LIN {X 0,Y 516.566,Z 410.559,A -85,B 0,C 180,E1 -4941.393,E2 -4941.393} C_VEL
LIN {X 0,Y 516.57,Z 414.408,A -85,B 0,C 180,E1 -4943.752,E2 -4943.752} C_VEL
LIN {X 0,Y 516.545,Z 418.324,A -85,B 0,C 180,E1 -4946.099,E2 -4946.099} C_VEL
LIN {X 0,Y 516.317,Z 423.538,A -85,B 0,C 180,E1 -4949.22,E2 -4949.22} C_VEL
LIN {X 0,Y 516.297,Z 425.129,A -85,B 0,C 180,E1 -4950.171,E2 -4950.171} C_VEL
LIN {X 0,Y 518.462,Z 437.532,A -85,B 0,C 180,E1 -4950.558,E2 -4950.558} C_VEL
LIN {X 0,Y 518.207,Z 449.848,A -85,B 0,C 180,E1 -4951.02,E2 -4951.02} C_VEL
LIN {X 0,Y 517.896,Z 462.254,A -85,B 0,C 180,E1 -4951.653,E2 -4951.653} C_VEL
LIN {X 0,Y 517.582,Z 473.862,A -85,B 0,C 180,E1 -4952.432,E2 -4952.432} C_VEL
LIN {X 0,Y 517.269,Z 484.296,A -85,B 0,C 180,E1 -4953.31,E2 -4953.31} C_VEL
LIN {X 0,Y 516.987,Z 493.731,A -85,B 0,C 180,E1 -4954.288,E2 -4954.288} C_VEL
LIN {X 0,Y 516.67,Z 502.845,A -85,B 0,C 180,E1 -4955.464,E2 -4955.464} C_VEL
LIN {X 0,Y 516.567,Z 510.483,A -85,B 0,C 180,E1 -4956.696,E2 -4956.696} C_VEL
LIN {X 0,Y 516.434,Z 516.081,A -85,B 0,C 180,E1 -4957.821,E2 -4957.821} C_VEL
LIN {X 0,Y 516.324,Z 520.76,A -85,B 0,C 180,E1 -4959.006,E2 -4959.006} C_VEL
LIN {X 0,Y 516.299,Z 524.331,A -85,B 0,C 180,E1 -4960.193,E2 -4960.193} C_VEL
LIN {X 0,Y 516.255,Z 526.976,A -85,B 0,C 180,E1 -4961.43,E2 -4961.43} C_VEL
LIN {X 0,Y 516.177,Z 528.494,A -85,B 0,C 180,E1 -4962.583,E2 -4962.583} C_VEL
LIN {X 0,Y 516.17,Z 529.065,A -85,B 0,C 180,E1 -4963.383,E2 -4963.383} C_VEL
LIN {X 0,Y 516.204,Z 528.984,A -85,B 0,C 180,E1 -4964.839,E2 -4964.839} C_VEL
LIN {X 0,Y 516.143,Z 528.194,A -85,B 0,C 180,E1 -4965.803,E2 -4965.803} C_VEL
LIN {X 0,Y 516.179,Z 527.062,A -85,B 0,C 180,E1 -4966.614,E2 -4966.614} C_VEL
LIN {X 0,Y 516.26,Z 524.946,A -85,B 0,C 180,E1 -4967.649,E2 -4967.649} C_VEL
LIN {X 0,Y 516.322,Z 520.828,A -85,B 0,C 180,E1 -4969.067,E2 -4969.067} C_VEL
LIN {X 0,Y 516.445,Z 515.75,A -85,B 0,C 180,E1 -4970.342,E2 -4970.342} C_VEL
LIN {X 0,Y 516.548,Z 509.6,A -85,B 0,C 180,E1 -4971.552,E2 -4971.552} C_VEL
LIN {X 0,Y 516.802,Z 501.624,A -85,B 0,C 180,E1 -4972.803,E2 -4972.803} C_VEL
LIN {X 0,Y 517.012,Z 493.278,A -85,B 0,C 180,E1 -4973.854,E2 -4973.854} C_VEL
LIN {X 0,Y 517.274,Z 482.922,A -85,B 0,C 180,E1 -4974.909,E2 -4974.909} C_VEL
LIN {X 0,Y 517.61,Z 472.647,A -85,B 0,C 180,E1 -4975.752,E2 -4975.752} C_VEL
LIN {X 0,Y 517.966,Z 461.051,A -85,B 0,C 180,E1 -4976.505,E2 -4976.505} C_VEL
LIN {X 0,Y 518.207,Z 448.508,A -85,B 0,C 180,E1 -4977.131,E2 -4977.131} C_VEL
LIN {X 0,Y 518.335,Z 435.967,A -85,B 0,C 180,E1 -4977.586,E2 -4977.586} C_VEL
LIN {X 0,Y 516.302,Z 425.139,A -85,B 0,C 180,E1 -4977.915,E2 -4977.915} C_VEL
LIN {X 0,Y 516.366,Z 419.746,A -85,B 0,C 180,E1 -4981.144,E2 -4981.144} C_VEL
LIN {X 0,Y 516.392,Z 415.182,A -85,B 0,C 180,E1 -4983.917,E2 -4983.917} C_VEL
LIN {X 0,Y 516.494,Z 410.526,A -85,B 0,C 180,E1 -4986.777,E2 -4986.777} C_VEL
LIN {X 0,Y 516.58,Z 406.717,A -85,B 0,C 180,E1 -4989.152,E2 -4989.152} C_VEL
LIN {X 0,Y 516.61,Z 402.558,A -85,B 0,C 180,E1 -4991.804,E2 -4991.804} C_VEL
LIN {X 0,Y 516.733,Z 397.617,A -85,B 0,C 180,E1 -4995.01,E2 -4995.01} C_VEL
LIN {X 0,Y 516.804,Z 392.843,A -85,B 0,C 180,E1 -4998.214,E2 -4998.214} C_VEL
LIN {X 0,Y 516.775,Z 391.335,A -85,B 0,C 180,E1 -4999.248,E2 -4999.248} C_VEL
LIN {X 0,Y 516.873,Z 391.102,A -85,B 0,C 180,E1 -5001.283,E2 -5001.283} C_VEL
LIN {X 0,Y 516.887,Z 391.102,A -85,B 0,C 180,E1 -5004.221,E2 -5004.221} C_VEL
LIN {X 0,Y 516.893,Z 391.101,A -85,B 0,C 180,E1 -5007.053,E2 -5007.053} C_VEL
LIN {X 0,Y 516.897,Z 391.102,A -85,B 0,C 180,E1 -5009.797,E2 -5009.797} C_VEL
LIN {X 0,Y 516.925,Z 391.097,A -85,B 0,C 180,E1 -5012.467,E2 -5012.467} C_VEL
LIN {X 0,Y 516.906,Z 391.097,A -85,B 0,C 180,E1 -5015.072,E2 -5015.072} C_VEL
LIN {X 0,Y 516.879,Z 391.102,A -85,B 0,C 180,E1 -5018.462,E2 -5018.462} C_VEL
LIN {X 0,Y 516.898,Z 391.097,A -85,B 0,C 180,E1 -5020.955,E2 -5020.955} C_VEL
LIN {X 0,Y 516.911,Z 391.097,A -85,B 0,C 180,E1 -5023.41,E2 -5023.41} C_VEL
LIN {X 0,Y 516.89,Z 391.1,A -85,B 0,C 180,E1 -5025.834,E2 -5025.834} C_VEL
LIN {X 0,Y 516.951,Z 391.094,A -85,B 0,C 180,E1 -5029.028,E2 -5029.028} C_VEL
LIN {X 0,Y 516.972,Z 391.092,A -85,B 0,C 180,E1 -5032.187,E2 -5032.187} C_VEL
LIN {X 0,Y 517.026,Z 391.082,A -85,B 0,C 180,E1 -5034.54,E2 -5034.54} C_VEL
LIN {X 0,Y 517.08,Z 391.075,A -85,B 0,C 180,E1 -5037.663,E2 -5037.663} C_VEL
LIN {X 0,Y 517.09,Z 391.075,A -85,B 0,C 180,E1 -5040.779,E2 -5040.779} C_VEL
LIN {X 0,Y 517.011,Z 391.083,A -85,B 0,C 180,E1 -5043.117,E2 -5043.117} C_VEL
LIN {X 0,Y 517.004,Z 391.084,A -85,B 0,C 180,E1 -5046.243,E2 -5046.243} C_VEL
LIN {X 0,Y 516.951,Z 391.091,A -85,B 0,C 180,E1 -5049.389,E2 -5049.389} C_VEL
LIN {X 0,Y 516.977,Z 391.089,A -85,B 0,C 180,E1 -5051.824,E2 -5051.824} C_VEL
LIN {X 0,Y 516.94,Z 391.092,A -85,B 0,C 180,E1 -5055.148,E2 -5055.148} C_VEL
LIN {X 0,Y 516.92,Z 391.095,A -85,B 0,C 180,E1 -5058.223,E2 -5058.223} C_VEL
LIN {X 0,Y 516.907,Z 391.099,A -85,B 0,C 180,E1 -5060.702,E2 -5060.702} C_VEL
LIN {X 0,Y 516.906,Z 391.097,A -85,B 0,C 180,E1 -5064.072,E2 -5064.072} C_VEL
LIN {X 0,Y 516.924,Z 391.097,A -85,B 0,C 180,E1 -5066.658,E2 -5066.658} C_VEL
LIN {X 0,Y 516.92,Z 391.099,A -85,B 0,C 180,E1 -5069.527,E2 -5069.527} C_VEL
LIN {X 0,Y 516.897,Z 391.101,A -85,B 0,C 180,E1 -5072.545,E2 -5072.545} C_VEL
LIN {X 0,Y 516.88,Z 391.103,A -85,B 0,C 180,E1 -5075.333,E2 -5075.333} C_VEL
LIN {X 0,Y 516.879,Z 391.098,A -85,B 0,C 180,E1 -5077.944,E2 -5077.944} C_VEL
LIN {X 0,Y 516.883,Z 391.099,A -85,B 0,C 180,E1 -5080.742,E2 -5080.742} C_VEL
LIN {X 0,Y 516.882,Z 391.103,A -85,B 0,C 180,E1 -5082.832,E2 -5082.832} C_VEL
LIN {X 0,Y 516.921,Z 391.095,A -85,B 0,C 180,E1 -5085.011,E2 -5085.011} C_VEL
LIN {X 0,Y 516.916,Z 391.097,A -85,B 0,C 180,E1 -5088.399,E2 -5088.399} C_VEL
LIN {X 0,Y 516.885,Z 391.102,A -85,B 0,C 180,E1 -5091.285,E2 -5091.285} C_VEL
LIN {X 0,Y 516.919,Z 391.214,A -85,B 0,C 180,E1 -5092.121,E2 -5092.121} C_VEL
LIN {X 0,Y 517.62,Z 395.743,A -85,B 0,C 180,E1 -5094.28,E2 -5094.28} C_VEL
LIN {X 0,Y 517.515,Z 401.084,A -85,B 0,C 180,E1 -5096.633,E2 -5096.633} C_VEL
LIN {X 0,Y 517.279,Z 407.585,A -85,B 0,C 180,E1 -5099.37,E2 -5099.37} C_VEL
LIN {X 0,Y 517.094,Z 414.221,A -85,B 0,C 180,E1 -5102.06,E2 -5102.06} C_VEL
LIN {X 0,Y 516.909,Z 421.933,A -85,B 0,C 180,E1 -5105.072,E2 -5105.072} C_VEL
LIN {X 0,Y 516.79,Z 429.804,A -85,B 0,C 180,E1 -5108.044,E2 -5108.044} C_VEL
LIN {X 0,Y 516.641,Z 437.65,A -85,B 0,C 180,E1 -5110.945,E2 -5110.945} C_VEL
LIN {X 0,Y 516.523,Z 446.704,A -85,B 0,C 180,E1 -5114.209,E2 -5114.209} C_VEL
LIN {X 0,Y 516.475,Z 451.986,A -85,B 0,C 180,E1 -5116.098,E2 -5116.098} C_VEL
LIN {X 0,Y 518.485,Z 465.419,A -85,B 0,C 180,E1 -5116.478,E2 -5116.478} C_VEL
LIN {X 0,Y 518.177,Z 478.753,A -85,B 0,C 180,E1 -5116.969,E2 -5116.969} C_VEL
LIN {X 0,Y 517.869,Z 491.25,A -85,B 0,C 180,E1 -5117.602,E2 -5117.602} C_VEL
LIN {X 0,Y 517.608,Z 502.486,A -85,B 0,C 180,E1 -5118.348,E2 -5118.348} C_VEL
LIN {X 0,Y 517.294,Z 513.161,A -85,B 0,C 180,E1 -5119.233,E2 -5119.233} C_VEL
LIN {X 0,Y 516.975,Z 522.78,A -85,B 0,C 180,E1 -5120.216,E2 -5120.216} C_VEL
LIN {X 0,Y 516.772,Z 530.667,A -85,B 0,C 180,E1 -5121.199,E2 -5121.199} C_VEL
LIN {X 0,Y 516.563,Z 538.368,A -85,B 0,C 180,E1 -5122.377,E2 -5122.377} C_VEL
LIN {X 0,Y 516.427,Z 545.468,A -85,B 0,C 180,E1 -5123.75,E2 -5123.75} C_VEL
LIN {X 0,Y 516.313,Z 550.19,A -85,B 0,C 180,E1 -5124.924,E2 -5124.924} C_VEL
LIN {X 0,Y 516.355,Z 553.802,A -85,B 0,C 180,E1 -5126.098,E2 -5126.098} C_VEL
LIN {X 0,Y 516.282,Z 555.661,A -85,B 0,C 180,E1 -5126.879,E2 -5126.879} C_VEL
LIN {X 0,Y 516.261,Z 557.057,A -85,B 0,C 180,E1 -5127.659,E2 -5127.659} C_VEL
LIN {X 0,Y 516.16,Z 558.658,A -85,B 0,C 180,E1 -5129.22,E2 -5129.22} C_VEL
LIN {X 0,Y 516.154,Z 558.875,A -85,B 0,C 180,E1 -5130,E2 -5130} C_VEL
LIN {X 0,Y 516.192,Z 558.054,A -85,B 0,C 180,E1 -5131.56,E2 -5131.56} C_VEL
LIN {X 0,Y 516.261,Z 557.061,A -85,B 0,C 180,E1 -5132.34,E2 -5132.34} C_VEL
LIN {X 0,Y 516.282,Z 555.667,A -85,B 0,C 180,E1 -5133.121,E2 -5133.121} C_VEL
LIN {X 0,Y 516.326,Z 552.734,A -85,B 0,C 180,E1 -5134.293,E2 -5134.293} C_VEL
LIN {X 0,Y 516.383,Z 548.763,A -85,B 0,C 180,E1 -5135.467,E2 -5135.467} C_VEL
LIN {X 0,Y 516.465,Z 543.474,A -85,B 0,C 180,E1 -5136.678,E2 -5136.678} C_VEL
LIN {X 0,Y 516.597,Z 537.215,A -85,B 0,C 180,E1 -5137.819,E2 -5137.819} C_VEL
LIN {X 0,Y 516.807,Z 529.187,A -85,B 0,C 180,E1 -5138.997,E2 -5138.997} C_VEL
LIN {X 0,Y 517.031,Z 521.006,A -85,B 0,C 180,E1 -5139.98,E2 -5139.98} C_VEL
LIN {X 0,Y 517.382,Z 511.032,A -85,B 0,C 180,E1 -5140.962,E2 -5140.962} C_VEL
LIN {X 0,Y 517.647,Z 501.193,A -85,B 0,C 180,E1 -5141.75,E2 -5141.75} C_VEL
LIN {X 0,Y 517.931,Z 490.039,A -85,B 0,C 180,E1 -5142.466,E2 -5142.466} C_VEL
LIN {X 0,Y 518.193,Z 477.64,A -85,B 0,C 180,E1 -5143.08,E2 -5143.08} C_VEL
LIN {X 0,Y 518.464,Z 464.605,A -85,B 0,C 180,E1 -5143.547,E2 -5143.547} C_VEL
LIN {X 0,Y 516.474,Z 452.021,A -85,B 0,C 180,E1 -5143.901,E2 -5143.901} C_VEL
LIN {X 0,Y 516.539,Z 444.499,A -85,B 0,C 180,E1 -5146.602,E2 -5146.602} C_VEL
LIN {X 0,Y 516.689,Z 436.591,A -85,B 0,C 180,E1 -5149.465,E2 -5149.465} C_VEL
LIN {X 0,Y 516.798,Z 428.734,A -85,B 0,C 180,E1 -5152.381,E2 -5152.381} C_VEL
LIN {X 0,Y 516.939,Z 420.899,A -85,B 0,C 180,E1 -5155.356,E2 -5155.356} C_VEL
LIN {X 0,Y 517.164,Z 413.088,A -85,B 0,C 180,E1 -5158.4,E2 -5158.4} C_VEL
LIN {X 0,Y 517.294,Z 406.262,A -85,B 0,C 180,E1 -5161.138,E2 -5161.138} C_VEL
LIN {X 0,Y 517.513,Z 399.174,A -85,B 0,C 180,E1 -5164.065,E2 -5164.065} C_VEL
LIN {X 0,Y 517.547,Z 395.297,A -85,B 0,C 180,E1 -5165.725,E2 -5165.725} C_VEL
LIN {X 0,Y 516.881,Z 391.103,A -85,B 0,C 180,E1 -5167.662,E2 -5167.662} C_VEL
LIN {X 0,Y 516.883,Z 391.103,A -85,B 0,C 180,E1 -5170.74,E2 -5170.74} C_VEL
LIN {X 0,Y 516.902,Z 391.101,A -85,B 0,C 180,E1 -5172.828,E2 -5172.828} C_VEL
LIN {X 0,Y 516.919,Z 391.098,A -85,B 0,C 180,E1 -5175.009,E2 -5175.009} C_VEL
LIN {X 0,Y 516.913,Z 391.096,A -85,B 0,C 180,E1 -5178.397,E2 -5178.397} C_VEL
LIN {X 0,Y 516.878,Z 391.098,A -85,B 0,C 180,E1 -5181.284,E2 -5181.284} C_VEL
LIN {X 0,Y 516.886,Z 391.1,A -85,B 0,C 180,E1 -5184.221,E2 -5184.221} C_VEL
LIN {X 0,Y 516.892,Z 391.096,A -85,B 0,C 180,E1 -5187.053,E2 -5187.053} C_VEL
LIN {X 0,Y 516.895,Z 391.097,A -85,B 0,C 180,E1 -5189.796,E2 -5189.796} C_VEL
LIN {X 0,Y 516.921,Z 391.097,A -85,B 0,C 180,E1 -5192.467,E2 -5192.467} C_VEL
LIN {X 0,Y 516.903,Z 391.094,A -85,B 0,C 180,E1 -5195.071,E2 -5195.071} C_VEL
LIN {X 0,Y 516.861,Z 391.103,A -85,B 0,C 180,E1 -5197.621,E2 -5197.621} C_VEL
LIN {X 0,Y 516.924,Z 391.098,A -85,B 0,C 180,E1 -5200.129,E2 -5200.129} C_VEL
LIN {X 0,Y 516.923,Z 391.093,A -85,B 0,C 180,E1 -5202.596,E2 -5202.596} C_VEL
LIN {X 0,Y 516.933,Z 391.091,A -85,B 0,C 180,E1 -5205.03,E2 -5205.03} C_VEL
LIN {X 0,Y 516.956,Z 391.09,A -85,B 0,C 180,E1 -5208.233,E2 -5208.233} C_VEL
LIN {X 0,Y 516.963,Z 391.092,A -85,B 0,C 180,E1 -5211.399,E2 -5211.399} C_VEL
LIN {X 0,Y 517.036,Z 391.078,A -85,B 0,C 180,E1 -5214.54,E2 -5214.54} C_VEL
LIN {X 0,Y 517.076,Z 391.077,A -85,B 0,C 180,E1 -5217.663,E2 -5217.663} C_VEL
LIN {X 0,Y 517.087,Z 391.074,A -85,B 0,C 180,E1 -5220.779,E2 -5220.779} C_VEL
LIN {X 0,Y 517.01,Z 391.086,A -85,B 0,C 180,E1 -5223.117,E2 -5223.117} C_VEL
LIN {X 0,Y 517.002,Z 391.082,A -85,B 0,C 180,E1 -5226.243,E2 -5226.243} C_VEL
LIN {X 0,Y 516.95,Z 391.091,A -85,B 0,C 180,E1 -5229.389,E2 -5229.389} C_VEL
LIN {X 0,Y 516.948,Z 391.089,A -85,B 0,C 180,E1 -5231.811,E2 -5231.811} C_VEL
LIN {X 0,Y 516.937,Z 391.093,A -85,B 0,C 180,E1 -5235.148,E2 -5235.148} C_VEL
LIN {X 0,Y 516.917,Z 391.096,A -85,B 0,C 180,E1 -5238.222,E2 -5238.222} C_VEL
LIN {X 0,Y 516.906,Z 391.098,A -85,B 0,C 180,E1 -5240.702,E2 -5240.702} C_VEL
LIN {X 0,Y 516.883,Z 391.097,A -85,B 0,C 180,E1 -5243.223,E2 -5243.223} C_VEL
LIN {X 0,Y 516.936,Z 391.096,A -85,B 0,C 180,E1 -5246.197,E2 -5246.197} C_VEL
LIN {X 0,Y 516.928,Z 391.091,A -85,B 0,C 180,E1 -5249.304,E2 -5249.304} C_VEL
LIN {X 0,Y 516.894,Z 391.098,A -85,B 0,C 180,E1 -5252.545,E2 -5252.545} C_VEL
LIN {X 0,Y 516.877,Z 391.098,A -85,B 0,C 180,E1 -5255.333,E2 -5255.333} C_VEL
LIN {X 0,Y 516.875,Z 391.104,A -85,B 0,C 180,E1 -5257.944,E2 -5257.944} C_VEL
LIN {X 0,Y 516.898,Z 391.094,A -85,B 0,C 180,E1 -5260.74,E2 -5260.74} C_VEL
LIN {X 0,Y 516.877,Z 391.102,A -85,B 0,C 180,E1 -5263.904,E2 -5263.904} C_VEL
LIN {X 0,Y 516.877,Z 391.099,A -85,B 0,C 180,E1 -5266.107,E2 -5266.107} C_VEL
LIN {X 0,Y 516.9,Z 391.098,A -85,B 0,C 180,E1 -5269.261,E2 -5269.261} C_VEL
LIN {X 0,Y 516.897,Z 391.094,A -85,B 0,C 180,E1 -5270.311,E2 -5270.311} C_VEL
LIN {X 0,Y 516.217,Z 391.181,A -85,B 0,C 180,E1 -5270.961,E2 -5270.961} C_VEL
LIN {X 0,Y 513.363,Z 391.54,A -85,B 0,C 180,E1 -5272.017,E2 -5272.017} C_VEL
LIN {X 0,Y 510.955,Z 391.843,A -85,B 0,C 180,E1 -5272.867,E2 -5272.867} C_VEL
LIN {X 0,Y 509.916,Z 391.97,A -85,B 0,C 180,E1 -5273.523,E2 -5273.523} C_VEL
LIN {X 0,Y 509.828,Z 391.978,A -85,B 0,C 180,E1 -5273.746,E2 -5273.746} C_VEL
LIN {X 0,Y 509.861,Z 391.97,A -85,B 0,C 180,E1 -5276.54,E2 -5276.54} C_VEL
LIN {X 0,Y 509.844,Z 391.979,A -85,B 0,C 180,E1 -5279.335,E2 -5279.335} C_VEL
LIN {X 0,Y 509.893,Z 391.966,A -85,B 0,C 180,E1 -5282.055,E2 -5282.055} C_VEL
LIN {X 0,Y 509.877,Z 391.972,A -85,B 0,C 180,E1 -5284.705,E2 -5284.705} C_VEL
LIN {X 0,Y 509.827,Z 391.977,A -85,B 0,C 180,E1 -5287.458,E2 -5287.458} C_VEL
LIN {X 0,Y 509.719,Z 391.996,A -85,B 0,C 180,E1 -5288.993,E2 -5288.993} C_VEL
LIN {X 0,Y 509.7,Z 396.598,A -85,B 0,C 180,E1 -5292.065,E2 -5292.065} C_VEL
LIN {X 0,Y 509.623,Z 400.933,A -85,B 0,C 180,E1 -5294.871,E2 -5294.871} C_VEL
LIN {X 0,Y 509.62,Z 406.261,A -85,B 0,C 180,E1 -5298.276,E2 -5298.276} C_VEL
LIN {X 0,Y 509.505,Z 411.037,A -85,B 0,C 180,E1 -5301.273,E2 -5301.273} C_VEL
LIN {X 0,Y 509.522,Z 414.894,A -85,B 0,C 180,E1 -5303.665,E2 -5303.665} C_VEL
LIN {X 0,Y 509.465,Z 418.811,A -85,B 0,C 180,E1 -5306.045,E2 -5306.045} C_VEL
LIN {X 0,Y 509.223,Z 425.214,A -85,B 0,C 180,E1 -5309.901,E2 -5309.901} C_VEL
LIN {X 0,Y 509.225,Z 425.336,A -85,B 0,C 180,E1 -5309.975,E2 -5309.975} C_VEL
LIN {X 0,Y 511.577,Z 438.331,A -85,B 0,C 180,E1 -5310.394,E2 -5310.394} C_VEL
LIN {X 0,Y 511.283,Z 451.056,A -85,B 0,C 180,E1 -5310.886,E2 -5310.886} C_VEL
LIN {X 0,Y 510.972,Z 462.377,A -85,B 0,C 180,E1 -5311.478,E2 -5311.478} C_VEL
LIN {X 0,Y 510.626,Z 474.008,A -85,B 0,C 180,E1 -5312.268,E2 -5312.268} C_VEL
LIN {X 0,Y 510.289,Z 484.452,A -85,B 0,C 180,E1 -5313.158,E2 -5313.158} C_VEL
LIN {X 0,Y 509.97,Z 493.899,A -85,B 0,C 180,E1 -5314.149,E2 -5314.149} C_VEL
LIN {X 0,Y 509.692,Z 501.66,A -85,B 0,C 180,E1 -5315.142,E2 -5315.142} C_VEL
LIN {X 0,Y 509.576,Z 509.233,A -85,B 0,C 180,E1 -5316.335,E2 -5316.335} C_VEL
LIN {X 0,Y 509.411,Z 515.357,A -85,B 0,C 180,E1 -5317.531,E2 -5317.531} C_VEL
LIN {X 0,Y 509.268,Z 520.232,A -85,B 0,C 180,E1 -5318.731,E2 -5318.731} C_VEL
LIN {X 0,Y 509.221,Z 523.986,A -85,B 0,C 180,E1 -5319.934,E2 -5319.934} C_VEL
LIN {X 0,Y 509.169,Z 527.327,A -85,B 0,C 180,E1 -5321.477,E2 -5321.477} C_VEL
LIN {X 0,Y 509.098,Z 528.892,A -85,B 0,C 180,E1 -5322.76,E2 -5322.76} C_VEL
LIN {X 0,Y 509.08,Z 529.322,A -85,B 0,C 180,E1 -5323.573,E2 -5323.573} C_VEL
LIN {X 0,Y 509.119,Z 529.147,A -85,B 0,C 180,E1 -5324.918,E2 -5324.918} C_VEL
LIN {X 0,Y 509.049,Z 528.168,A -85,B 0,C 180,E1 -5326.029,E2 -5326.029} C_VEL
LIN {X 0,Y 509.105,Z 526.898,A -85,B 0,C 180,E1 -5326.852,E2 -5326.852} C_VEL
LIN {X 0,Y 509.193,Z 524.272,A -85,B 0,C 180,E1 -5328.051,E2 -5328.051} C_VEL
LIN {X 0,Y 509.276,Z 520.304,A -85,B 0,C 180,E1 -5329.341,E2 -5329.341} C_VEL
LIN {X 0,Y 509.374,Z 515.381,A -85,B 0,C 180,E1 -5330.557,E2 -5330.557} C_VEL
LIN {X 0,Y 509.576,Z 508.653,A -85,B 0,C 180,E1 -5331.862,E2 -5331.862} C_VEL
LIN {X 0,Y 509.782,Z 501.855,A -85,B 0,C 180,E1 -5332.921,E2 -5332.921} C_VEL
LIN {X 0,Y 510.024,Z 493.519,A -85,B 0,C 180,E1 -5333.985,E2 -5333.985} C_VEL
LIN {X 0,Y 510.282,Z 483.897,A -85,B 0,C 180,E1 -5334.987,E2 -5334.987} C_VEL
LIN {X 0,Y 510.651,Z 472.899,A -85,B 0,C 180,E1 -5335.91,E2 -5335.91} C_VEL
LIN {X 0,Y 511.009,Z 462.159,A -85,B 0,C 180,E1 -5336.625,E2 -5336.625} C_VEL
LIN {X 0,Y 511.296,Z 450.036,A -85,B 0,C 180,E1 -5337.251,E2 -5337.251} C_VEL
LIN {X 0,Y 511.463,Z 437.14,A -85,B 0,C 180,E1 -5337.741,E2 -5337.741} C_VEL
LIN {X 0,Y 509.228,Z 425.355,A -85,B 0,C 180,E1 -5338.111,E2 -5338.111} C_VEL
LIN {X 0,Y 509.29,Z 420.272,A -85,B 0,C 180,E1 -5341.177,E2 -5341.177} C_VEL
LIN {X 0,Y 509.326,Z 416.481,A -85,B 0,C 180,E1 -5343.5,E2 -5343.5} C_VEL
LIN {X 0,Y 509.402,Z 411.826,A -85,B 0,C 180,E1 -5346.387,E2 -5346.387} C_VEL
LIN {X 0,Y 509.514,Z 407.023,A -85,B 0,C 180,E1 -5349.427,E2 -5349.427} C_VEL
LIN {X 0,Y 509.588,Z 402.249,A -85,B 0,C 180,E1 -5352.514,E2 -5352.514} C_VEL
LIN {X 0,Y 509.675,Z 398.031,A -85,B 0,C 180,E1 -5355.312,E2 -5355.312} C_VEL
LIN {X 0,Y 509.761,Z 393.906,A -85,B 0,C 180,E1 -5358.114,E2 -5358.114} C_VEL
LIN {X 0,Y 509.751,Z 391.992,A -85,B 0,C 180,E1 -5359.61,E2 -5359.61} C_VEL
LIN {X 0,Y 509.846,Z 391.978,A -85,B 0,C 180,E1 -5361.786,E2 -5361.786} C_VEL
LIN {X 0,Y 509.842,Z 391.979,A -85,B 0,C 180,E1 -5364.623,E2 -5364.623} C_VEL
LIN {X 0,Y 509.86,Z 391.975,A -85,B 0,C 180,E1 -5367.481,E2 -5367.481} C_VEL
LIN {X 0,Y 509.876,Z 391.972,A -85,B 0,C 180,E1 -5370.269,E2 -5370.269} C_VEL
LIN {X 0,Y 509.882,Z 391.974,A -85,B 0,C 180,E1 -5372.944,E2 -5372.944} C_VEL
LIN {X 0,Y 509.864,Z 391.978,A -85,B 0,C 180,E1 -5375.574,E2 -5375.574} C_VEL
LIN {X 0,Y 509.815,Z 391.979,A -85,B 0,C 180,E1 -5378.148,E2 -5378.148} C_VEL
LIN {X 0,Y 509.858,Z 391.974,A -85,B 0,C 180,E1 -5380.681,E2 -5380.681} C_VEL
LIN {X 0,Y 509.881,Z 391.975,A -85,B 0,C 180,E1 -5383.175,E2 -5383.175} C_VEL
LIN {X 0,Y 509.858,Z 391.974,A -85,B 0,C 180,E1 -5385.634,E2 -5385.634} C_VEL
LIN {X 0,Y 509.911,Z 391.97,A -85,B 0,C 180,E1 -5388.875,E2 -5388.875} C_VEL
LIN {X 0,Y 509.945,Z 391.968,A -85,B 0,C 180,E1 -5392.078,E2 -5392.078} C_VEL
LIN {X 0,Y 509.977,Z 391.959,A -85,B 0,C 180,E1 -5394.464,E2 -5394.464} C_VEL
LIN {X 0,Y 510.051,Z 391.951,A -85,B 0,C 180,E1 -5397.631,E2 -5397.631} C_VEL
LIN {X 0,Y 510.06,Z 391.951,A -85,B 0,C 180,E1 -5400.79,E2 -5400.79} C_VEL
LIN {X 0,Y 509.953,Z 391.962,A -85,B 0,C 180,E1 -5403.16,E2 -5403.16} C_VEL
LIN {X 0,Y 509.972,Z 391.96,A -85,B 0,C 180,E1 -5406.33,E2 -5406.33} C_VEL
LIN {X 0,Y 509.912,Z 391.97,A -85,B 0,C 180,E1 -5408.72,E2 -5408.72} C_VEL
LIN {X 0,Y 509.945,Z 391.964,A -85,B 0,C 180,E1 -5411.931,E2 -5411.931} C_VEL
LIN {X 0,Y 509.887,Z 391.971,A -85,B 0,C 180,E1 -5415.242,E2 -5415.242} C_VEL
LIN {X 0,Y 509.883,Z 391.972,A -85,B 0,C 180,E1 -5418.001,E2 -5418.001} C_VEL
LIN {X 0,Y 509.845,Z 391.977,A -85,B 0,C 180,E1 -5421.002,E2 -5421.002} C_VEL
LIN {X 0,Y 509.831,Z 391.982,A -85,B 0,C 180,E1 -5423.564,E2 -5423.564} C_VEL
LIN {X 0,Y 509.909,Z 391.973,A -85,B 0,C 180,E1 -5426.38,E2 -5426.38} C_VEL
LIN {X 0,Y 509.881,Z 391.972,A -85,B 0,C 180,E1 -5428.844,E2 -5428.844} C_VEL
LIN {X 0,Y 509.822,Z 391.979,A -85,B 0,C 180,E1 -5431.59,E2 -5431.59} C_VEL
LIN {X 0,Y 509.85,Z 391.975,A -85,B 0,C 180,E1 -5434.414,E2 -5434.414} C_VEL
LIN {X 0,Y 509.816,Z 391.978,A -85,B 0,C 180,E1 -5437.341,E2 -5437.341} C_VEL
LIN {X 0,Y 509.836,Z 391.977,A -85,B 0,C 180,E1 -5440.383,E2 -5440.383} C_VEL
LIN {X 0,Y 509.822,Z 391.982,A -85,B 0,C 180,E1 -5443.063,E2 -5443.063} C_VEL
LIN {X 0,Y 509.829,Z 391.982,A -85,B 0,C 180,E1 -5445.793,E2 -5445.793} C_VEL
LIN {X 0,Y 509.858,Z 391.978,A -85,B 0,C 180,E1 -5448.576,E2 -5448.576} C_VEL
LIN {X 0,Y 509.869,Z 392.014,A -85,B 0,C 180,E1 -5451.854,E2 -5451.854} C_VEL
LIN {X 0,Y 510.628,Z 397.059,A -85,B 0,C 180,E1 -5454.296,E2 -5454.296} C_VEL
LIN {X 0,Y 510.53,Z 402.155,A -85,B 0,C 180,E1 -5456.589,E2 -5456.589} C_VEL
LIN {X 0,Y 510.273,Z 408.627,A -85,B 0,C 180,E1 -5459.363,E2 -5459.363} C_VEL
LIN {X 0,Y 510.056,Z 415.196,A -85,B 0,C 180,E1 -5462.065,E2 -5462.065} C_VEL
LIN {X 0,Y 509.881,Z 421.819,A -85,B 0,C 180,E1 -5464.705,E2 -5464.705} C_VEL
LIN {X 0,Y 509.727,Z 429.017,A -85,B 0,C 180,E1 -5467.486,E2 -5467.486} C_VEL
LIN {X 0,Y 509.607,Z 436.363,A -85,B 0,C 180,E1 -5470.253,E2 -5470.253} C_VEL
LIN {X 0,Y 509.471,Z 445.359,A -85,B 0,C 180,E1 -5473.573,E2 -5473.573} C_VEL
LIN {X 0,Y 509.378,Z 451.771,A -85,B 0,C 180,E1 -5475.901,E2 -5475.901} C_VEL
LIN {X 0,Y 511.564,Z 465.965,A -85,B 0,C 180,E1 -5476.317,E2 -5476.317} C_VEL
LIN {X 0,Y 511.252,Z 478.534,A -85,B 0,C 180,E1 -5476.789,E2 -5476.789} C_VEL
LIN {X 0,Y 510.928,Z 491.083,A -85,B 0,C 180,E1 -5477.434,E2 -5477.434} C_VEL
LIN {X 0,Y 510.617,Z 502.27,A -85,B 0,C 180,E1 -5478.186,E2 -5478.186} C_VEL
LIN {X 0,Y 510.309,Z 512.947,A -85,B 0,C 180,E1 -5479.084,E2 -5479.084} C_VEL
LIN {X 0,Y 509.939,Z 522.566,A -85,B 0,C 180,E1 -5480.08,E2 -5480.08} C_VEL
LIN {X 0,Y 509.711,Z 530.454,A -85,B 0,C 180,E1 -5481.076,E2 -5481.076} C_VEL
LIN {X 0,Y 509.514,Z 538.158,A -85,B 0,C 180,E1 -5482.271,E2 -5482.271} C_VEL
LIN {X 0,Y 509.328,Z 545.259,A -85,B 0,C 180,E1 -5483.662,E2 -5483.662} C_VEL
LIN {X 0,Y 509.245,Z 549.983,A -85,B 0,C 180,E1 -5484.853,E2 -5484.853} C_VEL
LIN {X 0,Y 509.25,Z 553.594,A -85,B 0,C 180,E1 -5486.043,E2 -5486.043} C_VEL
LIN {X 0,Y 509.2,Z 555.456,A -85,B 0,C 180,E1 -5486.835,E2 -5486.835} C_VEL
LIN {X 0,Y 509.19,Z 556.852,A -85,B 0,C 180,E1 -5487.627,E2 -5487.627} C_VEL
LIN {X 0,Y 509.073,Z 558.454,A -85,B 0,C 180,E1 -5489.209,E2 -5489.209} C_VEL
LIN {X 0,Y 509.065,Z 558.671,A -85,B 0,C 180,E1 -5490,E2 -5490} C_VEL
LIN {X 0,Y 509.113,Z 557.851,A -85,B 0,C 180,E1 -5491.582,E2 -5491.582} C_VEL
LIN {X 0,Y 509.19,Z 556.859,A -85,B 0,C 180,E1 -5492.373,E2 -5492.373} C_VEL
LIN {X 0,Y 509.2,Z 555.464,A -85,B 0,C 180,E1 -5493.165,E2 -5493.165} C_VEL
LIN {X 0,Y 509.216,Z 552.53,A -85,B 0,C 180,E1 -5494.353,E2 -5494.353} C_VEL
LIN {X 0,Y 509.305,Z 548.559,A -85,B 0,C 180,E1 -5495.543,E2 -5495.543} C_VEL
LIN {X 0,Y 509.402,Z 542.904,A -85,B 0,C 180,E1 -5496.844,E2 -5496.844} C_VEL
LIN {X 0,Y 509.572,Z 535.773,A -85,B 0,C 180,E1 -5498.127,E2 -5498.127} C_VEL
LIN {X 0,Y 509.792,Z 527.489,A -85,B 0,C 180,E1 -5499.322,E2 -5499.322} C_VEL
LIN {X 0,Y 510.055,Z 518.999,A -85,B 0,C 180,E1 -5500.318,E2 -5500.318} C_VEL
LIN {X 0,Y 510.423,Z 508.509,A -85,B 0,C 180,E1 -5501.315,E2 -5501.315} C_VEL
LIN {X 0,Y 510.695,Z 497.211,A -85,B 0,C 180,E1 -5502.179,E2 -5502.179} C_VEL
LIN {X 0,Y 511.069,Z 486.757,A -85,B 0,C 180,E1 -5502.811,E2 -5502.811} C_VEL
LIN {X 0,Y 511.378,Z 475.089,A -85,B 0,C 180,E1 -5503.359,E2 -5503.359} C_VEL
LIN {X 0,Y 511.379,Z 463.931,A -85,B 0,C 180,E1 -5503.751,E2 -5503.751} C_VEL
LIN {X 0,Y 509.378,Z 451.815,A -85,B 0,C 180,E1 -5504.099,E2 -5504.099} C_VEL
LIN {X 0,Y 509.467,Z 444.292,A -85,B 0,C 180,E1 -5506.839,E2 -5506.839} C_VEL
LIN {X 0,Y 509.613,Z 436.431,A -85,B 0,C 180,E1 -5509.747,E2 -5509.747} C_VEL
LIN {X 0,Y 509.753,Z 429.085,A -85,B 0,C 180,E1 -5512.521,E2 -5512.521} C_VEL
LIN {X 0,Y 509.885,Z 421.892,A -85,B 0,C 180,E1 -5515.295,E2 -5515.295} C_VEL
LIN {X 0,Y 510.103,Z 414.667,A -85,B 0,C 180,E1 -5518.143,E2 -5518.143} C_VEL
LIN {X 0,Y 510.229,Z 408.505,A -85,B 0,C 180,E1 -5520.639,E2 -5520.639} C_VEL
LIN {X 0,Y 510.429,Z 401.818,A -85,B 0,C 180,E1 -5523.418,E2 -5523.418} C_VEL
LIN {X 0,Y 510.542,Z 396.536,A -85,B 0,C 180,E1 -5525.69,E2 -5525.69} C_VEL
LIN {X 0,Y 509.844,Z 391.979,A -85,B 0,C 180,E1 -5527.836,E2 -5527.836} C_VEL
LIN {X 0,Y 509.838,Z 391.98,A -85,B 0,C 180,E1 -5530.697,E2 -5530.697} C_VEL
LIN {X 0,Y 509.823,Z 391.976,A -85,B 0,C 180,E1 -5533.57,E2 -5533.57} C_VEL
LIN {X 0,Y 509.822,Z 391.979,A -85,B 0,C 180,E1 -5536.428,E2 -5536.428} C_VEL
LIN {X 0,Y 509.836,Z 391.975,A -85,B 0,C 180,E1 -5539.301,E2 -5539.301} C_VEL
LIN {X 0,Y 509.846,Z 391.973,A -85,B 0,C 180,E1 -5541.785,E2 -5541.785} C_VEL
LIN {X 0,Y 509.842,Z 391.981,A -85,B 0,C 180,E1 -5544.623,E2 -5544.623} C_VEL
LIN {X 0,Y 509.86,Z 391.972,A -85,B 0,C 180,E1 -5547.481,E2 -5547.481} C_VEL
LIN {X 0,Y 509.875,Z 391.975,A -85,B 0,C 180,E1 -5550.268,E2 -5550.268} C_VEL
LIN {X 0,Y 509.878,Z 391.97,A -85,B 0,C 180,E1 -5552.944,E2 -5552.944} C_VEL
LIN {X 0,Y 509.862,Z 391.973,A -85,B 0,C 180,E1 -5555.573,E2 -5555.573} C_VEL
LIN {X 0,Y 509.814,Z 391.983,A -85,B 0,C 180,E1 -5558.148,E2 -5558.148} C_VEL
LIN {X 0,Y 509.857,Z 391.973,A -85,B 0,C 180,E1 -5560.681,E2 -5560.681} C_VEL
LIN {X 0,Y 509.879,Z 391.971,A -85,B 0,C 180,E1 -5563.174,E2 -5563.174} C_VEL
LIN {X 0,Y 509.856,Z 391.977,A -85,B 0,C 180,E1 -5565.634,E2 -5565.634} C_VEL
LIN {X 0,Y 509.904,Z 391.967,A -85,B 0,C 180,E1 -5568.874,E2 -5568.874} C_VEL
LIN {X 0,Y 509.943,Z 391.964,A -85,B 0,C 180,E1 -5572.078,E2 -5572.078} C_VEL
LIN {X 0,Y 509.986,Z 391.956,A -85,B 0,C 180,E1 -5574.464,E2 -5574.464} C_VEL
LIN {X 0,Y 510.047,Z 391.953,A -85,B 0,C 180,E1 -5577.631,E2 -5577.631} C_VEL
LIN {X 0,Y 510.057,Z 391.95,A -85,B 0,C 180,E1 -5580.789,E2 -5580.789} C_VEL
LIN {X 0,Y 509.953,Z 391.965,A -85,B 0,C 180,E1 -5583.16,E2 -5583.16} C_VEL
LIN {X 0,Y 509.97,Z 391.959,A -85,B 0,C 180,E1 -5586.33,E2 -5586.33} C_VEL
LIN {X 0,Y 509.911,Z 391.971,A -85,B 0,C 180,E1 -5588.72,E2 -5588.72} C_VEL
LIN {X 0,Y 509.896,Z 391.967,A -85,B 0,C 180,E1 -5591.932,E2 -5591.932} C_VEL
LIN {X 0,Y 509.884,Z 391.971,A -85,B 0,C 180,E1 -5595.242,E2 -5595.242} C_VEL
LIN {X 0,Y 509.879,Z 391.97,A -85,B 0,C 180,E1 -5598.001,E2 -5598.001} C_VEL
LIN {X 0,Y 509.849,Z 391.976,A -85,B 0,C 180,E1 -5601.002,E2 -5601.002} C_VEL
LIN {X 0,Y 509.842,Z 391.974,A -85,B 0,C 180,E1 -5603.563,E2 -5603.563} C_VEL
LIN {X 0,Y 509.905,Z 391.971,A -85,B 0,C 180,E1 -5606.38,E2 -5606.38} C_VEL
LIN {X 0,Y 509.878,Z 391.971,A -85,B 0,C 180,E1 -5608.844,E2 -5608.844} C_VEL
LIN {X 0,Y 509.819,Z 391.978,A -85,B 0,C 180,E1 -5611.59,E2 -5611.59} C_VEL
LIN {X 0,Y 509.848,Z 391.976,A -85,B 0,C 180,E1 -5614.414,E2 -5614.414} C_VEL
LIN {X 0,Y 509.813,Z 391.978,A -85,B 0,C 180,E1 -5617.341,E2 -5617.341} C_VEL
LIN {X 0,Y 509.855,Z 391.973,A -85,B 0,C 180,E1 -5620.38,E2 -5620.38} C_VEL
LIN {X 0,Y 509.834,Z 391.975,A -85,B 0,C 180,E1 -5623.065,E2 -5623.065} C_VEL
LIN {X 0,Y 509.826,Z 391.981,A -85,B 0,C 180,E1 -5625.793,E2 -5625.793} C_VEL
LIN {X 0,Y 509.861,Z 391.97,A -85,B 0,C 180,E1 -5628.576,E2 -5628.576} C_VEL
LIN {X 0,Y 509.848,Z 391.975,A -85,B 0,C 180,E1 -5631.787,E2 -5631.787} C_VEL
LIN {X 0,Y 509.828,Z 391.978,A -85,B 0,C 180,E1 -5633.746,E2 -5633.746} C_VEL
LIN {X 0,Y 509.163,Z 392.058,A -85,B 0,C 180,E1 -5634.405,E2 -5634.405} C_VEL
LIN {X 0,Y 506.345,Z 392.415,A -85,B 0,C 180,E1 -5635.477,E2 -5635.477} C_VEL
LIN {X 0,Y 503.951,Z 392.713,A -85,B 0,C 180,E1 -5636.341,E2 -5636.341} C_VEL
LIN {X 0,Y 502.903,Z 392.841,A -85,B 0,C 180,E1 -5637.007,E2 -5637.007} C_VEL
LIN {X 0,Y 502.806,Z 392.851,A -85,B 0,C 180,E1 -5637.233,E2 -5637.233} C_VEL
LIN {X 0,Y 502.812,Z 392.848,A -85,B 0,C 180,E1 -5640.066,E2 -5640.066} C_VEL
LIN {X 0,Y 502.834,Z 392.847,A -85,B 0,C 180,E1 -5642.534,E2 -5642.534} C_VEL
LIN {X 0,Y 502.828,Z 392.851,A -85,B 0,C 180,E1 -5645.299,E2 -5645.299} C_VEL
LIN {X 0,Y 502.76,Z 392.855,A -85,B 0,C 180,E1 -5647.826,E2 -5647.826} C_VEL
LIN {X 0,Y 502.697,Z 392.868,A -85,B 0,C 180,E1 -5648.686,E2 -5648.686} C_VEL
LIN {X 0,Y 502.688,Z 393.597,A -85,B 0,C 180,E1 -5649.543,E2 -5649.543} C_VEL
LIN {X 0,Y 502.643,Z 397.424,A -85,B 0,C 180,E1 -5652.086,E2 -5652.086} C_VEL
LIN {X 0,Y 502.583,Z 401.534,A -85,B 0,C 180,E1 -5654.77,E2 -5654.77} C_VEL
LIN {X 0,Y 502.555,Z 406.88,A -85,B 0,C 180,E1 -5658.214,E2 -5658.214} C_VEL
LIN {X 0,Y 502.436,Z 411.512,A -85,B 0,C 180,E1 -5661.149,E2 -5661.149} C_VEL
LIN {X 0,Y 502.451,Z 415.379,A -85,B 0,C 180,E1 -5663.575,E2 -5663.575} C_VEL
LIN {X 0,Y 502.39,Z 419.296,A -85,B 0,C 180,E1 -5665.989,E2 -5665.989} C_VEL
LIN {X 0,Y 502.154,Z 425.543,A -85,B 0,C 180,E1 -5669.775,E2 -5669.775} C_VEL
LIN {X 0,Y 504.669,Z 439.154,A -85,B 0,C 180,E1 -5670.225,E2 -5670.225} C_VEL
LIN {X 0,Y 504.369,Z 452.255,A -85,B 0,C 180,E1 -5670.749,E2 -5670.749} C_VEL
LIN {X 0,Y 503.989,Z 464.103,A -85,B 0,C 180,E1 -5671.398,E2 -5671.398} C_VEL
LIN {X 0,Y 503.639,Z 475.426,A -85,B 0,C 180,E1 -5672.199,E2 -5672.199} C_VEL
LIN {X 0,Y 503.287,Z 485.663,A -85,B 0,C 180,E1 -5673.102,E2 -5673.102} C_VEL
LIN {X 0,Y 502.952,Z 494.068,A -85,B 0,C 180,E1 -5674.006,E2 -5674.006} C_VEL
LIN {X 0,Y 502.625,Z 503.189,A -85,B 0,C 180,E1 -5675.215,E2 -5675.215} C_VEL
LIN {X 0,Y 502.474,Z 510.528,A -85,B 0,C 180,E1 -5676.425,E2 -5676.425} C_VEL
LIN {X 0,Y 502.318,Z 516.446,A -85,B 0,C 180,E1 -5677.638,E2 -5677.638} C_VEL
LIN {X 0,Y 502.177,Z 521.135,A -85,B 0,C 180,E1 -5678.856,E2 -5678.856} C_VEL
LIN {X 0,Y 502.154,Z 524.712,A -85,B 0,C 180,E1 -5680.075,E2 -5680.075} C_VEL
LIN {X 0,Y 502.093,Z 527.667,A -85,B 0,C 180,E1 -5681.531,E2 -5681.531} C_VEL
LIN {X 0,Y 501.994,Z 529.223,A -85,B 0,C 180,E1 -5682.944,E2 -5682.944} C_VEL
LIN {X 0,Y 502.004,Z 529.565,A -85,B 0,C 180,E1 -5683.768,E2 -5683.768} C_VEL
LIN {X 0,Y 502.023,Z 529.314,A -85,B 0,C 180,E1 -5684.994,E2 -5684.994} C_VEL
LIN {X 0,Y 501.986,Z 528.088,A -85,B 0,C 180,E1 -5686.26,E2 -5686.26} C_VEL
LIN {X 0,Y 502.042,Z 526.735,A -85,B 0,C 180,E1 -5687.096,E2 -5687.096} C_VEL
LIN {X 0,Y 502.108,Z 523.823,A -85,B 0,C 180,E1 -5688.356,E2 -5688.356} C_VEL
LIN {X 0,Y 502.239,Z 519.779,A -85,B 0,C 180,E1 -5689.623,E2 -5689.623} C_VEL
LIN {X 0,Y 502.355,Z 514.454,A -85,B 0,C 180,E1 -5690.9,E2 -5690.9} C_VEL
LIN {X 0,Y 502.575,Z 507.602,A -85,B 0,C 180,E1 -5692.183,E2 -5692.183} C_VEL
LIN {X 0,Y 502.837,Z 498.944,A -85,B 0,C 180,E1 -5693.474,E2 -5693.474} C_VEL
LIN {X 0,Y 503.156,Z 489.917,A -85,B 0,C 180,E1 -5694.553,E2 -5694.553} C_VEL
LIN {X 0,Y 503.456,Z 479.931,A -85,B 0,C 180,E1 -5695.52,E2 -5695.52} C_VEL
LIN {X 0,Y 503.883,Z 468.639,A -85,B 0,C 180,E1 -5696.396,E2 -5696.396} C_VEL
LIN {X 0,Y 504.209,Z 458.024,A -85,B 0,C 180,E1 -5697.05,E2 -5697.05} C_VEL
LIN {X 0,Y 504.515,Z 445.944,A -85,B 0,C 180,E1 -5697.619,E2 -5697.619} C_VEL
LIN {X 0,Y 504.49,Z 437.858,A -85,B 0,C 180,E1 -5697.916,E2 -5697.916} C_VEL
LIN {X 0,Y 502.157,Z 425.54,A -85,B 0,C 180,E1 -5698.331,E2 -5698.331} C_VEL
LIN {X 0,Y 502.216,Z 420.517,A -85,B 0,C 180,E1 -5701.391,E2 -5701.391} C_VEL
LIN {X 0,Y 502.251,Z 415.751,A -85,B 0,C 180,E1 -5704.352,E2 -5704.352} C_VEL
LIN {X 0,Y 502.387,Z 411.358,A -85,B 0,C 180,E1 -5707.119,E2 -5707.119} C_VEL
LIN {X 0,Y 502.446,Z 406.823,A -85,B 0,C 180,E1 -5710.047,E2 -5710.047} C_VEL
LIN {X 0,Y 502.56,Z 401.949,A -85,B 0,C 180,E1 -5713.253,E2 -5713.253} C_VEL
LIN {X 0,Y 502.676,Z 396.968,A -85,B 0,C 180,E1 -5716.636,E2 -5716.636} C_VEL
LIN {X 0,Y 502.728,Z 393.549,A -85,B 0,C 180,E1 -5719.016,E2 -5719.016} C_VEL
LIN {X 0,Y 502.728,Z 392.866,A -85,B 0,C 180,E1 -5720.253,E2 -5720.253} C_VEL
LIN {X 0,Y 502.774,Z 392.86,A -85,B 0,C 180,E1 -5723.053,E2 -5723.053} C_VEL
LIN {X 0,Y 502.803,Z 392.855,A -85,B 0,C 180,E1 -5726.006,E2 -5726.006} C_VEL
LIN {X 0,Y 502.794,Z 392.855,A -85,B 0,C 180,E1 -5728.857,E2 -5728.857} C_VEL
LIN {X 0,Y 502.84,Z 392.849,A -85,B 0,C 180,E1 -5731.704,E2 -5731.704} C_VEL
LIN {X 0,Y 502.836,Z 392.853,A -85,B 0,C 180,E1 -5734.324,E2 -5734.324} C_VEL
LIN {X 0,Y 502.792,Z 392.857,A -85,B 0,C 180,E1 -5737.298,E2 -5737.298} C_VEL
LIN {X 0,Y 502.819,Z 392.853,A -85,B 0,C 180,E1 -5740.4,E2 -5740.4} C_VEL
LIN {X 0,Y 502.83,Z 392.852,A -85,B 0,C 180,E1 -5742.932,E2 -5742.932} C_VEL
LIN {X 0,Y 502.839,Z 392.848,A -85,B 0,C 180,E1 -5745.429,E2 -5745.429} C_VEL
LIN {X 0,Y 502.874,Z 392.845,A -85,B 0,C 180,E1 -5748.717,E2 -5748.717} C_VEL
LIN {X 0,Y 502.896,Z 392.845,A -85,B 0,C 180,E1 -5751.967,E2 -5751.967} C_VEL
LIN {X 0,Y 502.933,Z 392.837,A -85,B 0,C 180,E1 -5754.387,E2 -5754.387} C_VEL
LIN {X 0,Y 503.02,Z 392.826,A -85,B 0,C 180,E1 -5757.598,E2 -5757.598} C_VEL
LIN {X 0,Y 503.02,Z 392.827,A -85,B 0,C 180,E1 -5760,E2 -5760} C_VEL
LIN {X 0,Y 503.019,Z 392.83,A -85,B 0,C 180,E1 -5762.402,E2 -5762.402} C_VEL
LIN {X 0,Y 502.933,Z 392.841,A -85,B 0,C 180,E1 -5765.614,E2 -5765.614} C_VEL
LIN {X 0,Y 502.896,Z 392.84,A -85,B 0,C 180,E1 -5768.034,E2 -5768.034} C_VEL
LIN {X 0,Y 502.886,Z 392.845,A -85,B 0,C 180,E1 -5771.283,E2 -5771.283} C_VEL
LIN {X 0,Y 502.846,Z 392.852,A -85,B 0,C 180,E1 -5774.571,E2 -5774.571} C_VEL
LIN {X 0,Y 502.856,Z 392.848,A -85,B 0,C 180,E1 -5777.907,E2 -5777.907} C_VEL
LIN {X 0,Y 502.823,Z 392.855,A -85,B 0,C 180,E1 -5780.537,E2 -5780.537} C_VEL
LIN {X 0,Y 502.791,Z 392.856,A -85,B 0,C 180,E1 -5783.041,E2 -5783.041} C_VEL
LIN {X 0,Y 502.837,Z 392.849,A -85,B 0,C 180,E1 -5785.676,E2 -5785.676} C_VEL
LIN {X 0,Y 502.838,Z 392.85,A -85,B 0,C 180,E1 -5788.373,E2 -5788.373} C_VEL
LIN {X 0,Y 502.793,Z 392.855,A -85,B 0,C 180,E1 -5791.5,E2 -5791.5} C_VEL
LIN {X 0,Y 502.802,Z 392.853,A -85,B 0,C 180,E1 -5794.445,E2 -5794.445} C_VEL
LIN {X 0,Y 502.778,Z 392.856,A -85,B 0,C 180,E1 -5797.179,E2 -5797.179} C_VEL
LIN {X 0,Y 502.785,Z 392.858,A -85,B 0,C 180,E1 -5800.016,E2 -5800.016} C_VEL
LIN {X 0,Y 502.8,Z 392.854,A -85,B 0,C 180,E1 -5802.2,E2 -5802.2} C_VEL
LIN {X 0,Y 502.799,Z 392.855,A -85,B 0,C 180,E1 -5805.469,E2 -5805.469} C_VEL
LIN {X 0,Y 502.829,Z 392.852,A -85,B 0,C 180,E1 -5807.865,E2 -5807.865} C_VEL
LIN {X 0,Y 502.805,Z 392.855,A -85,B 0,C 180,E1 -5811.025,E2 -5811.025} C_VEL
LIN {X 0,Y 502.855,Z 392.954,A -85,B 0,C 180,E1 -5811.652,E2 -5811.652} C_VEL
LIN {X 0,Y 503.626,Z 397.919,A -85,B 0,C 180,E1 -5814.12,E2 -5814.12} C_VEL
LIN {X 0,Y 503.57,Z 402.164,A -85,B 0,C 180,E1 -5816.066,E2 -5816.066} C_VEL
LIN {X 0,Y 503.246,Z 409.672,A -85,B 0,C 180,E1 -5819.354,E2 -5819.354} C_VEL
LIN {X 0,Y 503.033,Z 416.243,A -85,B 0,C 180,E1 -5822.102,E2 -5822.102} C_VEL
LIN {X 0,Y 502.806,Z 423.941,A -85,B 0,C 180,E1 -5825.208,E2 -5825.208} C_VEL
LIN {X 0,Y 502.632,Z 432.84,A -85,B 0,C 180,E1 -5828.682,E2 -5828.682} C_VEL
LIN {X 0,Y 502.472,Z 440.803,A -85,B 0,C 180,E1 -5831.699,E2 -5831.699} C_VEL
LIN {X 0,Y 502.353,Z 449.297,A -85,B 0,C 180,E1 -5834.868,E2 -5834.868} C_VEL
LIN {X 0,Y 502.33,Z 451.802,A -85,B 0,C 180,E1 -5835.712,E2 -5835.712} C_VEL
LIN {X 0,Y 504.446,Z 464.973,A -85,B 0,C 180,E1 -5836.094,E2 -5836.094} C_VEL
LIN {X 0,Y 504.43,Z 476.055,A -85,B 0,C 180,E1 -5836.505,E2 -5836.505} C_VEL
LIN {X 0,Y 504.041,Z 488.274,A -85,B 0,C 180,E1 -5837.109,E2 -5837.109} C_VEL
LIN {X 0,Y 503.766,Z 499.635,A -85,B 0,C 180,E1 -5837.842,E2 -5837.842} C_VEL
LIN {X 0,Y 503.353,Z 510.584,A -85,B 0,C 180,E1 -5838.728,E2 -5838.728} C_VEL
LIN {X 0,Y 502.969,Z 520.563,A -85,B 0,C 180,E1 -5839.738,E2 -5839.738} C_VEL
LIN {X 0,Y 502.672,Z 530.242,A -85,B 0,C 180,E1 -5840.95,E2 -5840.95} C_VEL
LIN {X 0,Y 502.432,Z 537.947,A -85,B 0,C 180,E1 -5842.161,E2 -5842.161} C_VEL
LIN {X 0,Y 502.236,Z 545.049,A -85,B 0,C 180,E1 -5843.572,E2 -5843.572} C_VEL
LIN {X 0,Y 502.178,Z 549.776,A -85,B 0,C 180,E1 -5844.781,E2 -5844.781} C_VEL
LIN {X 0,Y 502.144,Z 553.388,A -85,B 0,C 180,E1 -5845.987,E2 -5845.987} C_VEL
LIN {X 0,Y 502.121,Z 555.25,A -85,B 0,C 180,E1 -5846.79,E2 -5846.79} C_VEL
LIN {X 0,Y 502.092,Z 556.647,A -85,B 0,C 180,E1 -5847.593,E2 -5847.593} C_VEL
LIN {X 0,Y 501.99,Z 558.25,A -85,B 0,C 180,E1 -5849.198,E2 -5849.198} C_VEL
LIN {X 0,Y 501.98,Z 558.468,A -85,B 0,C 180,E1 -5850,E2 -5850} C_VEL
LIN {X 0,Y 502.036,Z 557.648,A -85,B 0,C 180,E1 -5851.604,E2 -5851.604} C_VEL
LIN {X 0,Y 502.092,Z 556.655,A -85,B 0,C 180,E1 -5852.406,E2 -5852.406} C_VEL
LIN {X 0,Y 502.121,Z 555.261,A -85,B 0,C 180,E1 -5853.209,E2 -5853.209} C_VEL
LIN {X 0,Y 502.112,Z 552.326,A -85,B 0,C 180,E1 -5854.415,E2 -5854.415} C_VEL
LIN {X 0,Y 502.228,Z 548.355,A -85,B 0,C 180,E1 -5855.621,E2 -5855.621} C_VEL
LIN {X 0,Y 502.332,Z 542.346,A -85,B 0,C 180,E1 -5857.011,E2 -5857.011} C_VEL
LIN {X 0,Y 502.501,Z 535.568,A -85,B 0,C 180,E1 -5858.242,E2 -5858.242} C_VEL
LIN {X 0,Y 502.754,Z 527.283,A -85,B 0,C 180,E1 -5859.454,E2 -5859.454} C_VEL
LIN {X 0,Y 503.042,Z 518.792,A -85,B 0,C 180,E1 -5860.464,E2 -5860.464} C_VEL
LIN {X 0,Y 503.43,Z 508.302,A -85,B 0,C 180,E1 -5861.474,E2 -5861.474} C_VEL
LIN {X 0,Y 503.717,Z 497.003,A -85,B 0,C 180,E1 -5862.35,E2 -5862.35} C_VEL
LIN {X 0,Y 504.135,Z 486.549,A -85,B 0,C 180,E1 -5862.99,E2 -5862.99} C_VEL
LIN {X 0,Y 504.448,Z 474.879,A -85,B 0,C 180,E1 -5863.546,E2 -5863.546} C_VEL
LIN {X 0,Y 504.504,Z 465.019,A -85,B 0,C 180,E1 -5863.904,E2 -5863.904} C_VEL
LIN {X 0,Y 502.315,Z 451.611,A -85,B 0,C 180,E1 -5864.302,E2 -5864.302} C_VEL
LIN {X 0,Y 502.42,Z 444.121,A -85,B 0,C 180,E1 -5867.082,E2 -5867.082} C_VEL
LIN {X 0,Y 502.577,Z 436.283,A -85,B 0,C 180,E1 -5870.035,E2 -5870.035} C_VEL
LIN {X 0,Y 502.705,Z 428.46,A -85,B 0,C 180,E1 -5873.044,E2 -5873.044} C_VEL
LIN {X 0,Y 502.901,Z 420.638,A -85,B 0,C 180,E1 -5876.117,E2 -5876.117} C_VEL
LIN {X 0,Y 503.149,Z 412.824,A -85,B 0,C 180,E1 -5879.266,E2 -5879.266} C_VEL
LIN {X 0,Y 503.336,Z 406.14,A -85,B 0,C 180,E1 -5882.044,E2 -5882.044} C_VEL
LIN {X 0,Y 503.573,Z 398.352,A -85,B 0,C 180,E1 -5885.392,E2 -5885.392} C_VEL
LIN {X 0,Y 502.859,Z 393.227,A -85,B 0,C 180,E1 -5887.751,E2 -5887.751} C_VEL
LIN {X 0,Y 502.807,Z 392.856,A -85,B 0,C 180,E1 -5887.952,E2 -5887.952} C_VEL
LIN {X 0,Y 502.818,Z 392.856,A -85,B 0,C 180,E1 -5891.065,E2 -5891.065} C_VEL
LIN {X 0,Y 502.786,Z 392.854,A -85,B 0,C 180,E1 -5894.338,E2 -5894.338} C_VEL
LIN {X 0,Y 502.783,Z 392.859,A -85,B 0,C 180,E1 -5896.769,E2 -5896.769} C_VEL
LIN {X 0,Y 502.815,Z 392.853,A -85,B 0,C 180,E1 -5899.004,E2 -5899.004} C_VEL
LIN {X 0,Y 502.789,Z 392.854,A -85,B 0,C 180,E1 -5902.045,E2 -5902.045} C_VEL
LIN {X 0,Y 502.805,Z 392.852,A -85,B 0,C 180,E1 -5905.034,E2 -5905.034} C_VEL
LIN {X 0,Y 502.782,Z 392.856,A -85,B 0,C 180,E1 -5907.915,E2 -5907.915} C_VEL
LIN {X 0,Y 502.832,Z 392.85,A -85,B 0,C 180,E1 -5910.713,E2 -5910.713} C_VEL
LIN {X 0,Y 502.855,Z 392.845,A -85,B 0,C 180,E1 -5913.439,E2 -5913.439} C_VEL
LIN {X 0,Y 502.784,Z 392.858,A -85,B 0,C 180,E1 -5916.086,E2 -5916.086} C_VEL
LIN {X 0,Y 502.775,Z 392.855,A -85,B 0,C 180,E1 -5918.688,E2 -5918.688} C_VEL
LIN {X 0,Y 502.822,Z 392.85,A -85,B 0,C 180,E1 -5921.248,E2 -5921.248} C_VEL
LIN {X 0,Y 502.815,Z 392.854,A -85,B 0,C 180,E1 -5923.767,E2 -5923.767} C_VEL
LIN {X 0,Y 502.823,Z 392.851,A -85,B 0,C 180,E1 -5926.254,E2 -5926.254} C_VEL
LIN {X 0,Y 502.868,Z 392.843,A -85,B 0,C 180,E1 -5928.716,E2 -5928.716} C_VEL
LIN {X 0,Y 502.893,Z 392.843,A -85,B 0,C 180,E1 -5931.966,E2 -5931.966} C_VEL
LIN {X 0,Y 502.94,Z 392.834,A -85,B 0,C 180,E1 -5934.386,E2 -5934.386} C_VEL
LIN {X 0,Y 503.017,Z 392.829,A -85,B 0,C 180,E1 -5937.598,E2 -5937.598} C_VEL
LIN {X 0,Y 503.017,Z 392.825,A -85,B 0,C 180,E1 -5940,E2 -5940} C_VEL
LIN {X 0,Y 503.017,Z 392.825,A -85,B 0,C 180,E1 -5942.402,E2 -5942.402} C_VEL
LIN {X 0,Y 502.939,Z 392.836,A -85,B 0,C 180,E1 -5945.613,E2 -5945.613} C_VEL
LIN {X 0,Y 502.893,Z 392.84,A -85,B 0,C 180,E1 -5948.033,E2 -5948.033} C_VEL
LIN {X 0,Y 502.873,Z 392.846,A -85,B 0,C 180,E1 -5951.283,E2 -5951.283} C_VEL
LIN {X 0,Y 502.843,Z 392.852,A -85,B 0,C 180,E1 -5954.571,E2 -5954.571} C_VEL
LIN {X 0,Y 502.853,Z 392.845,A -85,B 0,C 180,E1 -5957.907,E2 -5957.907} C_VEL
LIN {X 0,Y 502.821,Z 392.854,A -85,B 0,C 180,E1 -5960.537,E2 -5960.537} C_VEL
LIN {X 0,Y 502.798,Z 392.853,A -85,B 0,C 180,E1 -5963.04,E2 -5963.04} C_VEL
LIN {X 0,Y 502.834,Z 392.848,A -85,B 0,C 180,E1 -5965.676,E2 -5965.676} C_VEL
LIN {X 0,Y 502.835,Z 392.851,A -85,B 0,C 180,E1 -5968.373,E2 -5968.373} C_VEL
LIN {X 0,Y 502.79,Z 392.853,A -85,B 0,C 180,E1 -5971.5,E2 -5971.5} C_VEL
LIN {X 0,Y 502.8,Z 392.853,A -85,B 0,C 180,E1 -5974.445,E2 -5974.445} C_VEL
LIN {X 0,Y 502.774,Z 392.854,A -85,B 0,C 180,E1 -5977.179,E2 -5977.179} C_VEL
LIN {X 0,Y 502.82,Z 392.853,A -85,B 0,C 180,E1 -5980.012,E2 -5980.012} C_VEL
LIN {X 0,Y 502.824,Z 392.85,A -85,B 0,C 180,E1 -5982.203,E2 -5982.203} C_VEL
LIN {X 0,Y 502.796,Z 392.856,A -85,B 0,C 180,E1 -5985.469,E2 -5985.469} C_VEL
LIN {X 0,Y 502.831,Z 392.85,A -85,B 0,C 180,E1 -5987.865,E2 -5987.865} C_VEL
LIN {X 0,Y 502.806,Z 392.851,A -85,B 0,C 180,E1 -5991.025,E2 -5991.025} C_VEL
LIN {X 0,Y 502.782,Z 392.852,A -85,B 0,C 180,E1 -5994.168,E2 -5994.168} C_VEL
LIN {X 0,Y 502.806,Z 392.851,A -85,B 0,C 180,E1 -5997.233,E2 -5997.233} C_VEL
LIN {X 0,Y 502.107,Z 392.938,A -85,B 0,C 180,E1 -5997.901,E2 -5997.901} C_VEL
LIN {X 0,Y 499.241,Z 393.298,A -85,B 0,C 180,E1 -5998.987,E2 -5998.987} C_VEL
LIN {X 0,Y 496.845,Z 393.593,A -85,B 0,C 180,E1 -5999.862,E2 -5999.862} C_VEL
LIN {X 0,Y 495.829,Z 393.719,A -85,B 0,C 180,E1 -6000.538,E2 -6000.538} C_VEL
LIN {X 0,Y 495.752,Z 393.73,A -85,B 0,C 180,E1 -6000.766,E2 -6000.766} C_VEL
LIN {X 0,Y 495.798,Z 393.723,A -85,B 0,C 180,E1 -6003.933,E2 -6003.933} C_VEL
LIN {X 0,Y 495.76,Z 393.733,A -85,B 0,C 180,E1 -6007.139,E2 -6007.139} C_VEL
LIN {X 0,Y 495.619,Z 393.993,A -85,B 0,C 180,E1 -6009.237,E2 -6009.237} C_VEL
LIN {X 0,Y 495.609,Z 397.832,A -85,B 0,C 180,E1 -6011.822,E2 -6011.822} C_VEL
LIN {X 0,Y 495.507,Z 402.964,A -85,B 0,C 180,E1 -6015.209,E2 -6015.209} C_VEL
LIN {X 0,Y 495.46,Z 408.09,A -85,B 0,C 180,E1 -6018.546,E2 -6018.546} C_VEL
LIN {X 0,Y 495.335,Z 413.265,A -85,B 0,C 180,E1 -6021.843,E2 -6021.843} C_VEL
LIN {X 0,Y 495.269,Z 417.168,A -85,B 0,C 180,E1 -6024.3,E2 -6024.3} C_VEL
LIN {X 0,Y 495.254,Z 421.104,A -85,B 0,C 180,E1 -6026.746,E2 -6026.746} C_VEL
LIN {X 0,Y 495.091,Z 425.736,A -85,B 0,C 180,E1 -6029.568,E2 -6029.568} C_VEL
LIN {X 0,Y 497.549,Z 438.691,A -85,B 0,C 180,E1 -6030,E2 -6030} C_VEL
LIN {X 0,Y 497.579,Z 449.005,A -85,B 0,C 180,E1 -6030.405,E2 -6030.405} C_VEL
LIN {X 0,Y 497.209,Z 460.87,A -85,B 0,C 180,E1 -6031.013,E2 -6031.013} C_VEL
LIN {X 0,Y 496.849,Z 471.627,A -85,B 0,C 180,E1 -6031.723,E2 -6031.723} C_VEL
LIN {X 0,Y 496.43,Z 482.645,A -85,B 0,C 180,E1 -6032.637,E2 -6032.637} C_VEL
LIN {X 0,Y 496.021,Z 492.466,A -85,B 0,C 180,E1 -6033.656,E2 -6033.656} C_VEL
LIN {X 0,Y 495.649,Z 502.004,A -85,B 0,C 180,E1 -6034.88,E2 -6034.88} C_VEL
LIN {X 0,Y 495.469,Z 509.594,A -85,B 0,C 180,E1 -6036.107,E2 -6036.107} C_VEL
LIN {X 0,Y 495.309,Z 515.72,A -85,B 0,C 180,E1 -6037.337,E2 -6037.337} C_VEL
LIN {X 0,Y 495.117,Z 520.607,A -85,B 0,C 180,E1 -6038.571,E2 -6038.571} C_VEL
LIN {X 0,Y 495.043,Z 524.37,A -85,B 0,C 180,E1 -6039.809,E2 -6039.809} C_VEL
LIN {X 0,Y 495.011,Z 526.314,A -85,B 0,C 180,E1 -6040.636,E2 -6040.636} C_VEL
LIN {X 0,Y 495.006,Z 527.985,A -85,B 0,C 180,E1 -6041.579,E2 -6041.579} C_VEL
LIN {X 0,Y 494.916,Z 529.545,A -85,B 0,C 180,E1 -6043.133,E2 -6043.133} C_VEL
LIN {X 0,Y 494.913,Z 529.81,A -85,B 0,C 180,E1 -6043.97,E2 -6043.97} C_VEL
LIN {X 0,Y 494.94,Z 529.477,A -85,B 0,C 180,E1 -6045.076,E2 -6045.076} C_VEL
LIN {X 0,Y 494.898,Z 528.008,A -85,B 0,C 180,E1 -6046.5,E2 -6046.5} C_VEL
LIN {X 0,Y 495.017,Z 525.192,A -85,B 0,C 180,E1 -6047.968,E2 -6047.968} C_VEL
LIN {X 0,Y 495.15,Z 520.742,A -85,B 0,C 180,E1 -6049.484,E2 -6049.484} C_VEL
LIN {X 0,Y 495.289,Z 514.676,A -85,B 0,C 180,E1 -6050.995,E2 -6050.995} C_VEL
LIN {X 0,Y 495.55,Z 507.832,A -85,B 0,C 180,E1 -6052.295,E2 -6052.295} C_VEL
LIN {X 0,Y 495.814,Z 499.174,A -85,B 0,C 180,E1 -6053.605,E2 -6053.605} C_VEL
LIN {X 0,Y 496.156,Z 490.484,A -85,B 0,C 180,E1 -6054.664,E2 -6054.664} C_VEL
LIN {X 0,Y 496.504,Z 480.056,A -85,B 0,C 180,E1 -6055.689,E2 -6055.689} C_VEL
LIN {X 0,Y 496.963,Z 468.905,A -85,B 0,C 180,E1 -6056.566,E2 -6056.566} C_VEL
LIN {X 0,Y 497.305,Z 458.318,A -85,B 0,C 180,E1 -6057.228,E2 -6057.228} C_VEL
LIN {X 0,Y 497.611,Z 446.928,A -85,B 0,C 180,E1 -6057.779,E2 -6057.779} C_VEL
LIN {X 0,Y 497.586,Z 438.647,A -85,B 0,C 180,E1 -6058.092,E2 -6058.092} C_VEL
LIN {X 0,Y 495.083,Z 425.754,A -85,B 0,C 180,E1 -6058.53,E2 -6058.53} C_VEL
LIN {X 0,Y 495.149,Z 420.644,A -85,B 0,C 180,E1 -6061.679,E2 -6061.679} C_VEL
LIN {X 0,Y 495.21,Z 416.006,A -85,B 0,C 180,E1 -6064.6,E2 -6064.6} C_VEL
LIN {X 0,Y 495.345,Z 411.339,A -85,B 0,C 180,E1 -6067.595,E2 -6067.595} C_VEL
LIN {X 0,Y 495.415,Z 406.552,A -85,B 0,C 180,E1 -6070.734,E2 -6070.734} C_VEL
LIN {X 0,Y 495.53,Z 401.649,A -85,B 0,C 180,E1 -6074.023,E2 -6074.023} C_VEL
LIN {X 0,Y 495.645,Z 397.183,A -85,B 0,C 180,E1 -6077.108,E2 -6077.108} C_VEL
LIN {X 0,Y 495.669,Z 394.111,A -85,B 0,C 180,E1 -6079.291,E2 -6079.291} C_VEL
LIN {X 0,Y 495.705,Z 393.742,A -85,B 0,C 180,E1 -6080.357,E2 -6080.357} C_VEL
LIN {X 0,Y 495.73,Z 393.74,A -85,B 0,C 180,E1 -6083.456,E2 -6083.456} C_VEL
LIN {X 0,Y 495.756,Z 393.736,A -85,B 0,C 180,E1 -6086.435,E2 -6086.435} C_VEL
LIN {X 0,Y 495.752,Z 393.734,A -85,B 0,C 180,E1 -6089.313,E2 -6089.313} C_VEL
LIN {X 0,Y 495.777,Z 393.729,A -85,B 0,C 180,E1 -6092.109,E2 -6092.109} C_VEL
LIN {X 0,Y 495.783,Z 393.728,A -85,B 0,C 180,E1 -6094.833,E2 -6094.833} C_VEL
LIN {X 0,Y 495.744,Z 393.733,A -85,B 0,C 180,E1 -6097.495,E2 -6097.495} C_VEL
LIN {X 0,Y 495.766,Z 393.733,A -85,B 0,C 180,E1 -6100.11,E2 -6100.11} C_VEL
LIN {X 0,Y 495.781,Z 393.728,A -85,B 0,C 180,E1 -6102.681,E2 -6102.681} C_VEL
LIN {X 0,Y 495.783,Z 393.727,A -85,B 0,C 180,E1 -6105.217,E2 -6105.217} C_VEL
LIN {X 0,Y 495.848,Z 393.719,A -85,B 0,C 180,E1 -6108.555,E2 -6108.555} C_VEL
LIN {X 0,Y 495.867,Z 393.719,A -85,B 0,C 180,E1 -6111.852,E2 -6111.852} C_VEL
LIN {X 0,Y 495.89,Z 393.714,A -85,B 0,C 180,E1 -6114.307,E2 -6114.307} C_VEL
LIN {X 0,Y 495.989,Z 393.702,A -85,B 0,C 180,E1 -6117.564,E2 -6117.564} C_VEL
LIN {X 0,Y 495.991,Z 393.702,A -85,B 0,C 180,E1 -6120,E2 -6120} C_VEL
LIN {X 0,Y 495.988,Z 393.706,A -85,B 0,C 180,E1 -6122.436,E2 -6122.436} C_VEL
LIN {X 0,Y 495.89,Z 393.717,A -85,B 0,C 180,E1 -6125.694,E2 -6125.694} C_VEL
LIN {X 0,Y 495.867,Z 393.716,A -85,B 0,C 180,E1 -6128.148,E2 -6128.148} C_VEL
LIN {X 0,Y 495.867,Z 393.721,A -85,B 0,C 180,E1 -6131.445,E2 -6131.445} C_VEL
LIN {X 0,Y 495.788,Z 393.729,A -85,B 0,C 180,E1 -6134.783,E2 -6134.783} C_VEL
LIN {X 0,Y 495.783,Z 393.731,A -85,B 0,C 180,E1 -6137.319,E2 -6137.319} C_VEL
LIN {X 0,Y 495.773,Z 393.73,A -85,B 0,C 180,E1 -6139.89,E2 -6139.89} C_VEL
LIN {X 0,Y 495.76,Z 393.732,A -85,B 0,C 180,E1 -6142.863,E2 -6142.863} C_VEL
LIN {X 0,Y 495.795,Z 393.728,A -85,B 0,C 180,E1 -6146.068,E2 -6146.068} C_VEL
LIN {X 0,Y 495.776,Z 393.729,A -85,B 0,C 180,E1 -6148.815,E2 -6148.815} C_VEL
LIN {X 0,Y 495.755,Z 393.731,A -85,B 0,C 180,E1 -6151.727,E2 -6151.727} C_VEL
LIN {X 0,Y 495.773,Z 393.729,A -85,B 0,C 180,E1 -6154.696,E2 -6154.696} C_VEL
LIN {X 0,Y 495.728,Z 393.732,A -85,B 0,C 180,E1 -6157.562,E2 -6157.562} C_VEL
LIN {X 0,Y 495.764,Z 393.73,A -85,B 0,C 180,E1 -6160.7,E2 -6160.7} C_VEL
LIN {X 0,Y 495.732,Z 393.736,A -85,B 0,C 180,E1 -6164.002,E2 -6164.002} C_VEL
LIN {X 0,Y 495.732,Z 393.737,A -85,B 0,C 180,E1 -6167.118,E2 -6167.118} C_VEL
LIN {X 0,Y 495.758,Z 393.734,A -85,B 0,C 180,E1 -6169.953,E2 -6169.953} C_VEL
LIN {X 0,Y 495.77,Z 393.841,A -85,B 0,C 180,E1 -6171.411,E2 -6171.411} C_VEL
LIN {X 0,Y 496.554,Z 398.512,A -85,B 0,C 180,E1 -6173.78,E2 -6173.78} C_VEL
LIN {X 0,Y 496.589,Z 403.253,A -85,B 0,C 180,E1 -6176.012,E2 -6176.012} C_VEL
LIN {X 0,Y 496.233,Z 410.741,A -85,B 0,C 180,E1 -6179.346,E2 -6179.346} C_VEL
LIN {X 0,Y 495.985,Z 417.265,A -85,B 0,C 180,E1 -6182.122,E2 -6182.122} C_VEL
LIN {X 0,Y 495.766,Z 424.577,A -85,B 0,C 180,E1 -6185.131,E2 -6185.131} C_VEL
LIN {X 0,Y 495.588,Z 432.696,A -85,B 0,C 180,E1 -6188.364,E2 -6188.364} C_VEL
LIN {X 0,Y 495.395,Z 440.505,A -85,B 0,C 180,E1 -6191.386,E2 -6191.386} C_VEL
LIN {X 0,Y 495.291,Z 448.341,A -85,B 0,C 180,E1 -6194.36,E2 -6194.36} C_VEL
LIN {X 0,Y 495.231,Z 451.574,A -85,B 0,C 180,E1 -6195.502,E2 -6195.502} C_VEL
LIN {X 0,Y 497.388,Z 464.749,A -85,B 0,C 180,E1 -6195.893,E2 -6195.893} C_VEL
LIN {X 0,Y 497.652,Z 469.336,A -85,B 0,C 180,E1 -6196.057,E2 -6196.057} C_VEL
LIN {X 0,Y 497.291,Z 482.373,A -85,B 0,C 180,E1 -6196.619,E2 -6196.619} C_VEL
LIN {X 0,Y 496.917,Z 494.001,A -85,B 0,C 180,E1 -6197.292,E2 -6197.292} C_VEL
LIN {X 0,Y 496.562,Z 505.695,A -85,B 0,C 180,E1 -6198.158,E2 -6198.158} C_VEL
LIN {X 0,Y 496.125,Z 516.597,A -85,B 0,C 180,E1 -6199.182,E2 -6199.182} C_VEL
LIN {X 0,Y 495.762,Z 525.455,A -85,B 0,C 180,E1 -6200.206,E2 -6200.206} C_VEL
LIN {X 0,Y 495.497,Z 534.098,A -85,B 0,C 180,E1 -6201.435,E2 -6201.435} C_VEL
LIN {X 0,Y 495.274,Z 541.004,A -85,B 0,C 180,E1 -6202.663,E2 -6202.663} C_VEL
LIN {X 0,Y 495.157,Z 547.053,A -85,B 0,C 180,E1 -6204.018,E2 -6204.018} C_VEL
LIN {X 0,Y 495.016,Z 552.108,A -85,B 0,C 180,E1 -6205.521,E2 -6205.521} C_VEL
LIN {X 0,Y 495.042,Z 555.045,A -85,B 0,C 180,E1 -6206.745,E2 -6206.745} C_VEL
LIN {X 0,Y 494.998,Z 556.442,A -85,B 0,C 180,E1 -6207.559,E2 -6207.559} C_VEL
LIN {X 0,Y 494.963,Z 557.438,A -85,B 0,C 180,E1 -6208.373,E2 -6208.373} C_VEL
LIN {X 0,Y 494.898,Z 558.264,A -85,B 0,C 180,E1 -6210,E2 -6210} C_VEL
LIN {X 0,Y 494.963,Z 557.445,A -85,B 0,C 180,E1 -6211.627,E2 -6211.627} C_VEL
LIN {X 0,Y 494.998,Z 556.452,A -85,B 0,C 180,E1 -6212.441,E2 -6212.441} C_VEL
LIN {X 0,Y 495.042,Z 555.058,A -85,B 0,C 180,E1 -6213.255,E2 -6213.255} C_VEL
LIN {X 0,Y 495.016,Z 552.122,A -85,B 0,C 180,E1 -6214.478,E2 -6214.478} C_VEL
LIN {X 0,Y 495.149,Z 548.151,A -85,B 0,C 180,E1 -6215.702,E2 -6215.702} C_VEL
LIN {X 0,Y 495.257,Z 542.04,A -85,B 0,C 180,E1 -6217.132,E2 -6217.132} C_VEL
LIN {X 0,Y 495.447,Z 535.363,A -85,B 0,C 180,E1 -6218.36,E2 -6218.36} C_VEL
LIN {X 0,Y 495.724,Z 527.078,A -85,B 0,C 180,E1 -6219.589,E2 -6219.589} C_VEL
LIN {X 0,Y 496.027,Z 518.586,A -85,B 0,C 180,E1 -6220.614,E2 -6220.614} C_VEL
LIN {X 0,Y 496.455,Z 508.095,A -85,B 0,C 180,E1 -6221.638,E2 -6221.638} C_VEL
LIN {X 0,Y 496.775,Z 496.67,A -85,B 0,C 180,E1 -6222.535,E2 -6222.535} C_VEL
LIN {X 0,Y 497.195,Z 486.34,A -85,B 0,C 180,E1 -6223.175,E2 -6223.175} C_VEL
LIN {X 0,Y 497.534,Z 474.669,A -85,B 0,C 180,E1 -6223.738,E2 -6223.738} C_VEL
LIN {X 0,Y 497.616,Z 466.146,A -85,B 0,C 180,E1 -6224.055,E2 -6224.055} C_VEL
LIN {X 0,Y 495.471,Z 453.132,A -85,B 0,C 180,E1 -6224.464,E2 -6224.464} C_VEL
LIN {X 0,Y 495.236,Z 451.406,A -85,B 0,C 180,E1 -6224.51,E2 -6224.51} C_VEL
LIN {X 0,Y 495.354,Z 443.945,A -85,B 0,C 180,E1 -6227.334,E2 -6227.334} C_VEL
LIN {X 0,Y 495.553,Z 435.418,A -85,B 0,C 180,E1 -6230.606,E2 -6230.606} C_VEL
LIN {X 0,Y 495.709,Z 427.191,A -85,B 0,C 180,E1 -6233.832,E2 -6233.832} C_VEL
LIN {X 0,Y 495.886,Z 419.363,A -85,B 0,C 180,E1 -6236.969,E2 -6236.969} C_VEL
LIN {X 0,Y 496.124,Z 412.678,A -85,B 0,C 180,E1 -6239.722,E2 -6239.722} C_VEL
LIN {X 0,Y 496.312,Z 405.995,A -85,B 0,C 180,E1 -6242.553,E2 -6242.553} C_VEL
LIN {X 0,Y 496.548,Z 399.323,A -85,B 0,C 180,E1 -6245.471,E2 -6245.471} C_VEL
LIN {X 0,Y 495.973,Z 394.866,A -85,B 0,C 180,E1 -6247.539,E2 -6247.539} C_VEL
LIN {X 0,Y 495.756,Z 393.734,A -85,B 0,C 180,E1 -6248.137,E2 -6248.137} C_VEL
LIN {X 0,Y 495.76,Z 393.733,A -85,B 0,C 180,E1 -6251.293,E2 -6251.293} C_VEL
LIN {X 0,Y 495.733,Z 393.731,A -85,B 0,C 180,E1 -6254,E2 -6254} C_VEL
LIN {X 0,Y 495.73,Z 393.735,A -85,B 0,C 180,E1 -6257.117,E2 -6257.117} C_VEL
LIN {X 0,Y 495.754,Z 393.729,A -85,B 0,C 180,E1 -6259.952,E2 -6259.952} C_VEL
LIN {X 0,Y 495.726,Z 393.737,A -85,B 0,C 180,E1 -6262.552,E2 -6262.552} C_VEL
LIN {X 0,Y 495.78,Z 393.726,A -85,B 0,C 180,E1 -6265.457,E2 -6265.457} C_VEL
LIN {X 0,Y 495.753,Z 393.734,A -85,B 0,C 180,E1 -6268.363,E2 -6268.363} C_VEL
LIN {X 0,Y 495.783,Z 393.726,A -85,B 0,C 180,E1 -6271.506,E2 -6271.506} C_VEL
LIN {X 0,Y 495.783,Z 393.729,A -85,B 0,C 180,E1 -6273.932,E2 -6273.932} C_VEL
LIN {X 0,Y 495.757,Z 393.729,A -85,B 0,C 180,E1 -6277.137,E2 -6277.137} C_VEL
LIN {X 0,Y 495.764,Z 393.733,A -85,B 0,C 180,E1 -6280.109,E2 -6280.109} C_VEL
LIN {X 0,Y 495.779,Z 393.727,A -85,B 0,C 180,E1 -6282.681,E2 -6282.681} C_VEL
LIN {X 0,Y 495.781,Z 393.728,A -85,B 0,C 180,E1 -6285.217,E2 -6285.217} C_VEL
LIN {X 0,Y 495.842,Z 393.719,A -85,B 0,C 180,E1 -6288.554,E2 -6288.554} C_VEL
LIN {X 0,Y 495.865,Z 393.72,A -85,B 0,C 180,E1 -6291.852,E2 -6291.852} C_VEL
LIN {X 0,Y 495.896,Z 393.712,A -85,B 0,C 180,E1 -6294.306,E2 -6294.306} C_VEL
LIN {X 0,Y 495.986,Z 393.705,A -85,B 0,C 180,E1 -6297.564,E2 -6297.564} C_VEL
LIN {X 0,Y 495.989,Z 393.701,A -85,B 0,C 180,E1 -6300,E2 -6300} C_VEL
LIN {X 0,Y 495.986,Z 393.701,A -85,B 0,C 180,E1 -6302.436,E2 -6302.436} C_VEL
LIN {X 0,Y 495.895,Z 393.713,A -85,B 0,C 180,E1 -6305.693,E2 -6305.693} C_VEL
LIN {X 0,Y 495.865,Z 393.716,A -85,B 0,C 180,E1 -6308.148,E2 -6308.148} C_VEL
LIN {X 0,Y 495.846,Z 393.719,A -85,B 0,C 180,E1 -6311.445,E2 -6311.445} C_VEL
LIN {X 0,Y 495.785,Z 393.729,A -85,B 0,C 180,E1 -6314.783,E2 -6314.783} C_VEL
LIN {X 0,Y 495.78,Z 393.727,A -85,B 0,C 180,E1 -6317.319,E2 -6317.319} C_VEL
LIN {X 0,Y 495.769,Z 393.728,A -85,B 0,C 180,E1 -6319.89,E2 -6319.89} C_VEL
LIN {X 0,Y 495.756,Z 393.732,A -85,B 0,C 180,E1 -6322.863,E2 -6322.863} C_VEL
LIN {X 0,Y 495.792,Z 393.729,A -85,B 0,C 180,E1 -6326.068,E2 -6326.068} C_VEL
LIN {X 0,Y 495.772,Z 393.728,A -85,B 0,C 180,E1 -6328.815,E2 -6328.815} C_VEL
LIN {X 0,Y 495.752,Z 393.732,A -85,B 0,C 180,E1 -6331.727,E2 -6331.727} C_VEL
LIN {X 0,Y 495.77,Z 393.728,A -85,B 0,C 180,E1 -6334.696,E2 -6334.696} C_VEL
LIN {X 0,Y 495.726,Z 393.735,A -85,B 0,C 180,E1 -6337.562,E2 -6337.562} C_VEL
LIN {X 0,Y 495.787,Z 393.728,A -85,B 0,C 180,E1 -6340.053,E2 -6340.053} C_VEL
LIN {X 0,Y 495.758,Z 393.727,A -85,B 0,C 180,E1 -6342.88,E2 -6342.88} C_VEL
LIN {X 0,Y 495.732,Z 393.734,A -85,B 0,C 180,E1 -6346,E2 -6346} C_VEL
LIN {X 0,Y 495.764,Z 393.726,A -85,B 0,C 180,E1 -6348.706,E2 -6348.706} C_VEL
LIN {X 0,Y 495.751,Z 393.735,A -85,B 0,C 180,E1 -6351.41,E2 -6351.41} C_VEL
LIN {X 0,Y 495.755,Z 393.727,A -85,B 0,C 180,E1 -6354.464,E2 -6354.464} C_VEL
LIN {X 0,Y 495.767,Z 393.732,A -85,B 0,C 180,E1 -6357.407,E2 -6357.407} C_VEL
LIN {X 0,Y 495.764,Z 393.726,A -85,B 0,C 180,E1 -6360.254,E2 -6360.254} C_VEL
LIN {X 0,Y 495.752,Z 393.73,A -85,B 0,C 180,E1 -6360.766,E2 -6360.766} C_VEL
LIN {X 0,Y 495.097,Z 393.817,A -85,B 0,C 180,E1 -6361.445,E2 -6361.445} C_VEL
LIN {X 0,Y 492.244,Z 394.169,A -85,B 0,C 180,E1 -6362.548,E2 -6362.548} C_VEL
LIN {X 0,Y 489.836,Z 394.469,A -85,B 0,C 180,E1 -6363.437,E2 -6363.437} C_VEL
LIN {X 0,Y 488.819,Z 394.592,A -85,B 0,C 180,E1 -6364.123,E2 -6364.123} C_VEL
LIN {X 0,Y 488.746,Z 394.602,A -85,B 0,C 180,E1 -6364.356,E2 -6364.356} C_VEL
LIN {X 0,Y 488.723,Z 394.609,A -85,B 0,C 180,E1 -6367.154,E2 -6367.154} C_VEL
LIN {X 0,Y 488.57,Z 394.832,A -85,B 0,C 180,E1 -6369.23,E2 -6369.23} C_VEL
LIN {X 0,Y 488.523,Z 399.524,A -85,B 0,C 180,E1 -6372.416,E2 -6372.416} C_VEL
LIN {X 0,Y 488.453,Z 403.387,A -85,B 0,C 180,E1 -6374.99,E2 -6374.99} C_VEL
LIN {X 0,Y 488.42,Z 408.542,A -85,B 0,C 180,E1 -6378.379,E2 -6378.379} C_VEL
LIN {X 0,Y 488.283,Z 413.734,A -85,B 0,C 180,E1 -6381.725,E2 -6381.725} C_VEL
LIN {X 0,Y 488.213,Z 417.655,A -85,B 0,C 180,E1 -6384.217,E2 -6384.217} C_VEL
LIN {X 0,Y 488.2,Z 421.59,A -85,B 0,C 180,E1 -6386.699,E2 -6386.699} C_VEL
LIN {X 0,Y 488.027,Z 425.885,A -85,B 0,C 180,E1 -6389.356,E2 -6389.356} C_VEL
LIN {X 0,Y 490.669,Z 439.497,A -85,B 0,C 180,E1 -6389.821,E2 -6389.821} C_VEL
LIN {X 0,Y 490.633,Z 451.328,A -85,B 0,C 180,E1 -6390.308,E2 -6390.308} C_VEL
LIN {X 0,Y 490.235,Z 462.74,A -85,B 0,C 180,E1 -6390.924,E2 -6390.924} C_VEL
LIN {X 0,Y 489.813,Z 474.434,A -85,B 0,C 180,E1 -6391.747,E2 -6391.747} C_VEL
LIN {X 0,Y 489.386,Z 484.915,A -85,B 0,C 180,E1 -6392.675,E2 -6392.675} C_VEL
LIN {X 0,Y 488.971,Z 494.393,A -85,B 0,C 180,E1 -6393.708,E2 -6393.708} C_VEL
LIN {X 0,Y 488.571,Z 503.538,A -85,B 0,C 180,E1 -6394.951,E2 -6394.951} C_VEL
LIN {X 0,Y 488.403,Z 510.825,A -85,B 0,C 180,E1 -6396.185,E2 -6396.185} C_VEL
LIN {X 0,Y 488.228,Z 516.807,A -85,B 0,C 180,E1 -6397.444,E2 -6397.444} C_VEL
LIN {X 0,Y 488.029,Z 521.51,A -85,B 0,C 180,E1 -6398.697,E2 -6398.697} C_VEL
LIN {X 0,Y 487.957,Z 525.098,A -85,B 0,C 180,E1 -6399.953,E2 -6399.953} C_VEL
LIN {X 0,Y 487.91,Z 526.937,A -85,B 0,C 180,E1 -6400.793,E2 -6400.793} C_VEL
LIN {X 0,Y 487.927,Z 528.309,A -85,B 0,C 180,E1 -6401.634,E2 -6401.634} C_VEL
LIN {X 0,Y 487.839,Z 529.289,A -85,B 0,C 180,E1 -6402.48,E2 -6402.48} C_VEL
LIN {X 0,Y 487.812,Z 529.87,A -85,B 0,C 180,E1 -6403.327,E2 -6403.327} C_VEL
LIN {X 0,Y 487.834,Z 530.003,A -85,B 0,C 180,E1 -6404.176,E2 -6404.176} C_VEL
LIN {X 0,Y 487.861,Z 529.64,A -85,B 0,C 180,E1 -6405.163,E2 -6405.163} C_VEL
LIN {X 0,Y 487.811,Z 527.909,A -85,B 0,C 180,E1 -6406.747,E2 -6406.747} C_VEL
LIN {X 0,Y 487.939,Z 525.259,A -85,B 0,C 180,E1 -6408.08,E2 -6408.08} C_VEL
LIN {X 0,Y 488.058,Z 521.706,A -85,B 0,C 180,E1 -6409.341,E2 -6409.341} C_VEL
LIN {X 0,Y 488.193,Z 516.809,A -85,B 0,C 180,E1 -6410.653,E2 -6410.653} C_VEL
LIN {X 0,Y 488.374,Z 510.503,A -85,B 0,C 180,E1 -6411.972,E2 -6411.972} C_VEL
LIN {X 0,Y 488.727,Z 502.369,A -85,B 0,C 180,E1 -6413.321,E2 -6413.321} C_VEL
LIN {X 0,Y 489.036,Z 494.232,A -85,B 0,C 180,E1 -6414.404,E2 -6414.404} C_VEL
LIN {X 0,Y 489.375,Z 483.897,A -85,B 0,C 180,E1 -6415.52,E2 -6415.52} C_VEL
LIN {X 0,Y 489.845,Z 473.672,A -85,B 0,C 180,E1 -6416.408,E2 -6416.408} C_VEL
LIN {X 0,Y 490.217,Z 462.519,A -85,B 0,C 180,E1 -6417.183,E2 -6417.183} C_VEL
LIN {X 0,Y 490.629,Z 449.715,A -85,B 0,C 180,E1 -6417.861,E2 -6417.861} C_VEL
LIN {X 0,Y 490.764,Z 440.002,A -85,B 0,C 180,E1 -6418.251,E2 -6418.251} C_VEL
LIN {X 0,Y 488.208,Z 427.182,A -85,B 0,C 180,E1 -6418.698,E2 -6418.698} C_VEL
LIN {X 0,Y 488.021,Z 425.962,A -85,B 0,C 180,E1 -6418.74,E2 -6418.74} C_VEL
LIN {X 0,Y 488.087,Z 420.446,A -85,B 0,C 180,E1 -6422.192,E2 -6422.192} C_VEL
LIN {X 0,Y 488.153,Z 415.805,A -85,B 0,C 180,E1 -6425.161,E2 -6425.161} C_VEL
LIN {X 0,Y 488.3,Z 411.093,A -85,B 0,C 180,E1 -6428.234,E2 -6428.234} C_VEL
LIN {X 0,Y 488.398,Z 406.108,A -85,B 0,C 180,E1 -6431.559,E2 -6431.559} C_VEL
LIN {X 0,Y 488.498,Z 401.354,A -85,B 0,C 180,E1 -6434.825,E2 -6434.825} C_VEL
LIN {X 0,Y 488.613,Z 397.615,A -85,B 0,C 180,E1 -6437.466,E2 -6437.466} C_VEL
LIN {X 0,Y 488.63,Z 394.623,A -85,B 0,C 180,E1 -6439.666,E2 -6439.666} C_VEL
LIN {X 0,Y 488.674,Z 394.619,A -85,B 0,C 180,E1 -6442.278,E2 -6442.278} C_VEL
LIN {X 0,Y 488.724,Z 394.613,A -85,B 0,C 180,E1 -6445.051,E2 -6445.051} C_VEL
LIN {X 0,Y 488.701,Z 394.615,A -85,B 0,C 180,E1 -6448.045,E2 -6448.045} C_VEL
LIN {X 0,Y 488.728,Z 394.608,A -85,B 0,C 180,E1 -6450.73,E2 -6450.73} C_VEL
LIN {X 0,Y 488.761,Z 394.603,A -85,B 0,C 180,E1 -6453.528,E2 -6453.528} C_VEL
LIN {X 0,Y 488.687,Z 394.611,A -85,B 0,C 180,E1 -6456.254,E2 -6456.254} C_VEL
LIN {X 0,Y 488.739,Z 394.605,A -85,B 0,C 180,E1 -6459.175,E2 -6459.175} C_VEL
LIN {X 0,Y 488.728,Z 394.606,A -85,B 0,C 180,E1 -6462.423,E2 -6462.423} C_VEL
LIN {X 0,Y 488.755,Z 394.603,A -85,B 0,C 180,E1 -6465,E2 -6465} C_VEL
LIN {X 0,Y 488.801,Z 394.596,A -85,B 0,C 180,E1 -6468.388,E2 -6468.388} C_VEL
LIN {X 0,Y 488.812,Z 394.597,A -85,B 0,C 180,E1 -6471.734,E2 -6471.734} C_VEL
LIN {X 0,Y 488.849,Z 394.591,A -85,B 0,C 180,E1 -6474.224,E2 -6474.224} C_VEL
LIN {X 0,Y 488.956,Z 394.578,A -85,B 0,C 180,E1 -6477.529,E2 -6477.529} C_VEL
LIN {X 0,Y 488.97,Z 394.579,A -85,B 0,C 180,E1 -6480.824,E2 -6480.824} C_VEL
LIN {X 0,Y 488.955,Z 394.582,A -85,B 0,C 180,E1 -6482.472,E2 -6482.472} C_VEL
LIN {X 0,Y 488.85,Z 394.593,A -85,B 0,C 180,E1 -6485.776,E2 -6485.776} C_VEL
LIN {X 0,Y 488.812,Z 394.596,A -85,B 0,C 180,E1 -6488.267,E2 -6488.267} C_VEL
LIN {X 0,Y 488.826,Z 394.597,A -85,B 0,C 180,E1 -6491.612,E2 -6491.612} C_VEL
LIN {X 0,Y 488.759,Z 394.603,A -85,B 0,C 180,E1 -6495.001,E2 -6495.001} C_VEL
LIN {X 0,Y 488.749,Z 394.605,A -85,B 0,C 180,E1 -6498.443,E2 -6498.443} C_VEL
LIN {X 0,Y 488.702,Z 394.611,A -85,B 0,C 180,E1 -6501.071,E2 -6501.071} C_VEL
LIN {X 0,Y 488.688,Z 394.614,A -85,B 0,C 180,E1 -6503.746,E2 -6503.746} C_VEL
LIN {X 0,Y 488.794,Z 394.599,A -85,B 0,C 180,E1 -6506.946,E2 -6506.946} C_VEL
LIN {X 0,Y 488.715,Z 394.609,A -85,B 0,C 180,E1 -6510.365,E2 -6510.365} C_VEL
LIN {X 0,Y 488.732,Z 394.607,A -85,B 0,C 180,E1 -6513.485,E2 -6513.485} C_VEL
LIN {X 0,Y 488.685,Z 394.611,A -85,B 0,C 180,E1 -6516.356,E2 -6516.356} C_VEL
LIN {X 0,Y 488.699,Z 394.609,A -85,B 0,C 180,E1 -6519.255,E2 -6519.255} C_VEL
LIN {X 0,Y 488.706,Z 394.612,A -85,B 0,C 180,E1 -6521.601,E2 -6521.601} C_VEL
LIN {X 0,Y 488.71,Z 394.61,A -85,B 0,C 180,E1 -6524.802,E2 -6524.802} C_VEL
LIN {X 0,Y 488.693,Z 394.614,A -85,B 0,C 180,E1 -6527.476,E2 -6527.476} C_VEL
LIN {X 0,Y 488.732,Z 394.609,A -85,B 0,C 180,E1 -6529.677,E2 -6529.677} C_VEL
LIN {X 0,Y 488.738,Z 394.729,A -85,B 0,C 180,E1 -6531.165,E2 -6531.165} C_VEL
LIN {X 0,Y 489.507,Z 399.254,A -85,B 0,C 180,E1 -6533.515,E2 -6533.515} C_VEL
LIN {X 0,Y 489.593,Z 403.259,A -85,B 0,C 180,E1 -6535.458,E2 -6535.458} C_VEL
LIN {X 0,Y 489.322,Z 409.673,A -85,B 0,C 180,E1 -6538.397,E2 -6538.397} C_VEL
LIN {X 0,Y 489.051,Z 416.149,A -85,B 0,C 180,E1 -6541.237,E2 -6541.237} C_VEL
LIN {X 0,Y 488.787,Z 423.757,A -85,B 0,C 180,E1 -6544.447,E2 -6544.447} C_VEL
LIN {X 0,Y 488.555,Z 431.477,A -85,B 0,C 180,E1 -6547.592,E2 -6547.592} C_VEL
LIN {X 0,Y 488.405,Z 438.119,A -85,B 0,C 180,E1 -6550.236,E2 -6550.236} C_VEL
LIN {X 0,Y 488.253,Z 445.924,A -85,B 0,C 180,E1 -6553.269,E2 -6553.269} C_VEL
LIN {X 0,Y 488.171,Z 451.347,A -85,B 0,C 180,E1 -6555.288,E2 -6555.288} C_VEL
LIN {X 0,Y 490.258,Z 464.522,A -85,B 0,C 180,E1 -6555.683,E2 -6555.683} C_VEL
LIN {X 0,Y 490.762,Z 469.116,A -85,B 0,C 180,E1 -6555.857,E2 -6555.857} C_VEL
LIN {X 0,Y 490.412,Z 481.161,A -85,B 0,C 180,E1 -6556.375,E2 -6556.375} C_VEL
LIN {X 0,Y 489.998,Z 492.79,A -85,B 0,C 180,E1 -6557.043,E2 -6557.043} C_VEL
LIN {X 0,Y 489.622,Z 504.212,A -85,B 0,C 180,E1 -6557.882,E2 -6557.882} C_VEL
LIN {X 0,Y 489.246,Z 514.423,A -85,B 0,C 180,E1 -6558.818,E2 -6558.818} C_VEL
LIN {X 0,Y 488.789,Z 523.607,A -85,B 0,C 180,E1 -6559.855,E2 -6559.855} C_VEL
LIN {X 0,Y 488.482,Z 532.56,A -85,B 0,C 180,E1 -6561.103,E2 -6561.103} C_VEL
LIN {X 0,Y 488.243,Z 539.767,A -85,B 0,C 180,E1 -6562.348,E2 -6562.348} C_VEL
LIN {X 0,Y 488.081,Z 545.092,A -85,B 0,C 180,E1 -6563.49,E2 -6563.49} C_VEL
LIN {X 0,Y 488.027,Z 549.361,A -85,B 0,C 180,E1 -6564.629,E2 -6564.629} C_VEL
LIN {X 0,Y 487.934,Z 552.974,A -85,B 0,C 180,E1 -6565.87,E2 -6565.87} C_VEL
LIN {X 0,Y 487.965,Z 554.84,A -85,B 0,C 180,E1 -6566.697,E2 -6566.697} C_VEL
LIN {X 0,Y 487.891,Z 557.234,A -85,B 0,C 180,E1 -6568.349,E2 -6568.349} C_VEL
LIN {X 0,Y 487.819,Z 558.061,A -85,B 0,C 180,E1 -6570,E2 -6570} C_VEL
LIN {X 0,Y 487.891,Z 557.242,A -85,B 0,C 180,E1 -6571.651,E2 -6571.651} C_VEL
LIN {X 0,Y 487.965,Z 554.855,A -85,B 0,C 180,E1 -6573.302,E2 -6573.302} C_VEL
LIN {X 0,Y 487.927,Z 551.919,A -85,B 0,C 180,E1 -6574.544,E2 -6574.544} C_VEL
LIN {X 0,Y 488.052,Z 547.947,A -85,B 0,C 180,E1 -6575.785,E2 -6575.785} C_VEL
LIN {X 0,Y 488.184,Z 541.836,A -85,B 0,C 180,E1 -6577.236,E2 -6577.236} C_VEL
LIN {X 0,Y 488.381,Z 535.157,A -85,B 0,C 180,E1 -6578.482,E2 -6578.482} C_VEL
LIN {X 0,Y 488.691,Z 526.872,A -85,B 0,C 180,E1 -6579.728,E2 -6579.728} C_VEL
LIN {X 0,Y 489.03,Z 518.38,A -85,B 0,C 180,E1 -6580.767,E2 -6580.767} C_VEL
LIN {X 0,Y 489.478,Z 507.887,A -85,B 0,C 180,E1 -6581.806,E2 -6581.806} C_VEL
LIN {X 0,Y 489.844,Z 496.132,A -85,B 0,C 180,E1 -6582.739,E2 -6582.739} C_VEL
LIN {X 0,Y 490.328,Z 484.205,A -85,B 0,C 180,E1 -6583.468,E2 -6583.468} C_VEL
LIN {X 0,Y 490.693,Z 471.858,A -85,B 0,C 180,E1 -6584.039,E2 -6584.039} C_VEL
LIN {X 0,Y 490.589,Z 466.504,A -85,B 0,C 180,E1 -6584.24,E2 -6584.24} C_VEL
LIN {X 0,Y 488.4,Z 452.991,A -85,B 0,C 180,E1 -6584.677,E2 -6584.677} C_VEL
LIN {X 0,Y 488.157,Z 451.22,A -85,B 0,C 180,E1 -6584.726,E2 -6584.726} C_VEL
LIN {X 0,Y 488.285,Z 443.771,A -85,B 0,C 180,E1 -6587.593,E2 -6587.593} C_VEL
LIN {X 0,Y 488.502,Z 435.682,A -85,B 0,C 180,E1 -6590.748,E2 -6590.748} C_VEL
LIN {X 0,Y 488.659,Z 428.128,A -85,B 0,C 180,E1 -6593.747,E2 -6593.747} C_VEL
LIN {X 0,Y 488.845,Z 420.263,A -85,B 0,C 180,E1 -6596.955,E2 -6596.955} C_VEL
LIN {X 0,Y 489.084,Z 413.637,A -85,B 0,C 180,E1 -6599.719,E2 -6599.719} C_VEL
LIN {X 0,Y 489.311,Z 406.944,A -85,B 0,C 180,E1 -6602.588,E2 -6602.588} C_VEL
LIN {X 0,Y 489.536,Z 400.274,A -85,B 0,C 180,E1 -6605.55,E2 -6605.55} C_VEL
LIN {X 0,Y 488.908,Z 395.604,A -85,B 0,C 180,E1 -6607.756,E2 -6607.756} C_VEL
LIN {X 0,Y 488.747,Z 394.608,A -85,B 0,C 180,E1 -6608.324,E2 -6608.324} C_VEL
LIN {X 0,Y 488.72,Z 394.607,A -85,B 0,C 180,E1 -6611.601,E2 -6611.601} C_VEL
LIN {X 0,Y 488.708,Z 394.612,A -85,B 0,C 180,E1 -6614.8,E2 -6614.8} C_VEL
LIN {X 0,Y 488.691,Z 394.609,A -85,B 0,C 180,E1 -6617.474,E2 -6617.474} C_VEL
LIN {X 0,Y 488.728,Z 394.604,A -85,B 0,C 180,E1 -6619.676,E2 -6619.676} C_VEL
LIN {X 0,Y 488.677,Z 394.615,A -85,B 0,C 180,E1 -6622.841,E2 -6622.841} C_VEL
LIN {X 0,Y 488.73,Z 394.606,A -85,B 0,C 180,E1 -6625.887,E2 -6625.887} C_VEL
LIN {X 0,Y 488.69,Z 394.612,A -85,B 0,C 180,E1 -6628.82,E2 -6628.82} C_VEL
LIN {X 0,Y 488.74,Z 394.605,A -85,B 0,C 180,E1 -6631.671,E2 -6631.671} C_VEL
LIN {X 0,Y 488.74,Z 394.608,A -85,B 0,C 180,E1 -6634.444,E2 -6634.444} C_VEL
LIN {X 0,Y 488.72,Z 394.606,A -85,B 0,C 180,E1 -6637.153,E2 -6637.153} C_VEL
LIN {X 0,Y 488.717,Z 394.609,A -85,B 0,C 180,E1 -6639.81,E2 -6639.81} C_VEL
LIN {X 0,Y 488.726,Z 394.607,A -85,B 0,C 180,E1 -6642.423,E2 -6642.423} C_VEL
LIN {X 0,Y 488.753,Z 394.602,A -85,B 0,C 180,E1 -6644.999,E2 -6644.999} C_VEL
LIN {X 0,Y 488.796,Z 394.597,A -85,B 0,C 180,E1 -6648.387,E2 -6648.387} C_VEL
LIN {X 0,Y 488.809,Z 394.599,A -85,B 0,C 180,E1 -6651.733,E2 -6651.733} C_VEL
LIN {X 0,Y 488.854,Z 394.59,A -85,B 0,C 180,E1 -6654.224,E2 -6654.224} C_VEL
LIN {X 0,Y 488.953,Z 394.58,A -85,B 0,C 180,E1 -6657.528,E2 -6657.528} C_VEL
LIN {X 0,Y 488.96,Z 394.577,A -85,B 0,C 180,E1 -6660,E2 -6660} C_VEL
LIN {X 0,Y 488.954,Z 394.578,A -85,B 0,C 180,E1 -6662.471,E2 -6662.471} C_VEL
LIN {X 0,Y 488.853,Z 394.59,A -85,B 0,C 180,E1 -6665.776,E2 -6665.776} C_VEL
LIN {X 0,Y 488.81,Z 394.595,A -85,B 0,C 180,E1 -6668.266,E2 -6668.266} C_VEL
LIN {X 0,Y 488.799,Z 394.596,A -85,B 0,C 180,E1 -6671.612,E2 -6671.612} C_VEL
LIN {X 0,Y 488.755,Z 394.604,A -85,B 0,C 180,E1 -6675,E2 -6675} C_VEL
LIN {X 0,Y 488.746,Z 394.608,A -85,B 0,C 180,E1 -6678.442,E2 -6678.442} C_VEL
LIN {X 0,Y 488.704,Z 394.609,A -85,B 0,C 180,E1 -6681.071,E2 -6681.071} C_VEL
LIN {X 0,Y 488.693,Z 394.61,A -85,B 0,C 180,E1 -6683.745,E2 -6683.745} C_VEL
LIN {X 0,Y 488.791,Z 394.598,A -85,B 0,C 180,E1 -6686.946,E2 -6686.946} C_VEL
LIN {X 0,Y 488.711,Z 394.61,A -85,B 0,C 180,E1 -6690.365,E2 -6690.365} C_VEL
LIN {X 0,Y 488.729,Z 394.605,A -85,B 0,C 180,E1 -6693.485,E2 -6693.485} C_VEL
LIN {X 0,Y 488.682,Z 394.612,A -85,B 0,C 180,E1 -6696.356,E2 -6696.356} C_VEL
LIN {X 0,Y 488.742,Z 394.603,A -85,B 0,C 180,E1 -6699.25,E2 -6699.25} C_VEL
LIN {X 0,Y 488.729,Z 394.604,A -85,B 0,C 180,E1 -6702.521,E2 -6702.521} C_VEL
LIN {X 0,Y 488.697,Z 394.61,A -85,B 0,C 180,E1 -6705.976,E2 -6705.976} C_VEL
LIN {X 0,Y 488.72,Z 394.604,A -85,B 0,C 180,E1 -6708.587,E2 -6708.587} C_VEL
LIN {X 0,Y 488.736,Z 394.603,A -85,B 0,C 180,E1 -6710.943,E2 -6710.943} C_VEL
LIN {X 0,Y 488.682,Z 394.61,A -85,B 0,C 180,E1 -6713.869,E2 -6713.869} C_VEL
LIN {X 0,Y 488.737,Z 394.604,A -85,B 0,C 180,E1 -6716.878,E2 -6716.878} C_VEL
LIN {X 0,Y 488.722,Z 394.605,A -85,B 0,C 180,E1 -6719.781,E2 -6719.781} C_VEL
LIN {X 0,Y 488.797,Z 394.601,A -85,B 0,C 180,E1 -6723.055,E2 -6723.055} C_VEL
LIN {X 0,Y 488.746,Z 394.602,A -85,B 0,C 180,E1 -6724.356,E2 -6724.356} C_VEL
LIN {X 0,Y 488.101,Z 394.688,A -85,B 0,C 180,E1 -6725.043,E2 -6725.043} C_VEL
LIN {X 0,Y 485.237,Z 395.042,A -85,B 0,C 180,E1 -6726.16,E2 -6726.16} C_VEL
LIN {X 0,Y 482.78,Z 395.351,A -85,B 0,C 180,E1 -6727.059,E2 -6727.059} C_VEL
LIN {X 0,Y 481.698,Z 395.48,A -85,B 0,C 180,E1 -6727.755,E2 -6727.755} C_VEL
LIN {X 0,Y 481.597,Z 395.492,A -85,B 0,C 180,E1 -6727.99,E2 -6727.99} C_VEL
LIN {X 0,Y 481.519,Z 395.509,A -85,B 0,C 180,E1 -6729.085,E2 -6729.085} C_VEL
LIN {X 0,Y 481.482,Z 399.928,A -85,B 0,C 180,E1 -6732.15,E2 -6732.15} C_VEL
LIN {X 0,Y 481.405,Z 403.81,A -85,B 0,C 180,E1 -6734.765,E2 -6734.765} C_VEL
LIN {X 0,Y 481.379,Z 408.989,A -85,B 0,C 180,E1 -6738.206,E2 -6738.206} C_VEL
LIN {X 0,Y 481.216,Z 414.203,A -85,B 0,C 180,E1 -6741.602,E2 -6741.602} C_VEL
LIN {X 0,Y 481.159,Z 418.14,A -85,B 0,C 180,E1 -6744.132,E2 -6744.132} C_VEL
LIN {X 0,Y 481.148,Z 422.091,A -85,B 0,C 180,E1 -6746.651,E2 -6746.651} C_VEL
LIN {X 0,Y 480.939,Z 426.072,A -85,B 0,C 180,E1 -6749.137,E2 -6749.137} C_VEL
LIN {X 0,Y 483.763,Z 440.266,A -85,B 0,C 180,E1 -6749.636,E2 -6749.636} C_VEL
LIN {X 0,Y 483.769,Z 450.286,A -85,B 0,C 180,E1 -6750.052,E2 -6750.052} C_VEL
LIN {X 0,Y 483.32,Z 462.846,A -85,B 0,C 180,E1 -6750.729,E2 -6750.729} C_VEL
LIN {X 0,Y 482.959,Z 473.277,A -85,B 0,C 180,E1 -6751.459,E2 -6751.459} C_VEL
LIN {X 0,Y 482.451,Z 484.018,A -85,B 0,C 180,E1 -6752.4,E2 -6752.4} C_VEL
LIN {X 0,Y 481.975,Z 494.559,A -85,B 0,C 180,E1 -6753.553,E2 -6753.553} C_VEL
LIN {X 0,Y 481.55,Z 503.713,A -85,B 0,C 180,E1 -6754.814,E2 -6754.814} C_VEL
LIN {X 0,Y 481.342,Z 511.065,A -85,B 0,C 180,E1 -6756.077,E2 -6756.077} C_VEL
LIN {X 0,Y 481.138,Z 517.87,A -85,B 0,C 180,E1 -6757.554,E2 -6757.554} C_VEL
LIN {X 0,Y 480.952,Z 522.375,A -85,B 0,C 180,E1 -6758.826,E2 -6758.826} C_VEL
LIN {X 0,Y 480.877,Z 525.797,A -85,B 0,C 180,E1 -6760.101,E2 -6760.101} C_VEL
LIN {X 0,Y 480.842,Z 528.629,A -85,B 0,C 180,E1 -6761.686,E2 -6761.686} C_VEL
LIN {X 0,Y 480.751,Z 529.69,A -85,B 0,C 180,E1 -6762.667,E2 -6762.667} C_VEL
LIN {X 0,Y 480.712,Z 530.133,A -85,B 0,C 180,E1 -6763.528,E2 -6763.528} C_VEL
LIN {X 0,Y 480.732,Z 530.167,A -85,B 0,C 180,E1 -6764.39,E2 -6764.39} C_VEL
LIN {X 0,Y 480.751,Z 529.801,A -85,B 0,C 180,E1 -6765.256,E2 -6765.256} C_VEL
LIN {X 0,Y 480.703,Z 529.009,A -85,B 0,C 180,E1 -6766.128,E2 -6766.128} C_VEL
LIN {X 0,Y 480.731,Z 527.746,A -85,B 0,C 180,E1 -6767.001,E2 -6767.001} C_VEL
LIN {X 0,Y 480.858,Z 525.327,A -85,B 0,C 180,E1 -6768.193,E2 -6768.193} C_VEL
LIN {X 0,Y 480.997,Z 521.179,A -85,B 0,C 180,E1 -6769.637,E2 -6769.637} C_VEL
LIN {X 0,Y 481.185,Z 515.853,A -85,B 0,C 180,E1 -6771.021,E2 -6771.021} C_VEL
LIN {X 0,Y 481.391,Z 509.552,A -85,B 0,C 180,E1 -6772.308,E2 -6772.308} C_VEL
LIN {X 0,Y 481.691,Z 502.774,A -85,B 0,C 180,E1 -6773.427,E2 -6773.427} C_VEL
LIN {X 0,Y 482.038,Z 494.471,A -85,B 0,C 180,E1 -6774.552,E2 -6774.552} C_VEL
LIN {X 0,Y 482.397,Z 485.038,A -85,B 0,C 180,E1 -6775.596,E2 -6775.596} C_VEL
LIN {X 0,Y 482.923,Z 473.957,A -85,B 0,C 180,E1 -6776.583,E2 -6776.583} C_VEL
LIN {X 0,Y 483.337,Z 462.336,A -85,B 0,C 180,E1 -6777.399,E2 -6777.399} C_VEL
LIN {X 0,Y 483.74,Z 450.084,A -85,B 0,C 180,E1 -6778.057,E2 -6778.057} C_VEL
LIN {X 0,Y 483.832,Z 440.67,A -85,B 0,C 180,E1 -6778.446,E2 -6778.446} C_VEL
LIN {X 0,Y 481.196,Z 427.656,A -85,B 0,C 180,E1 -6778.915,E2 -6778.915} C_VEL
LIN {X 0,Y 480.957,Z 426.134,A -85,B 0,C 180,E1 -6778.979,E2 -6778.979} C_VEL
LIN {X 0,Y 481.029,Z 421.27,A -85,B 0,C 180,E1 -6782.07,E2 -6782.07} C_VEL
LIN {X 0,Y 481.106,Z 416.566,A -85,B 0,C 180,E1 -6785.11,E2 -6785.11} C_VEL
LIN {X 0,Y 481.222,Z 412.287,A -85,B 0,C 180,E1 -6787.941,E2 -6787.941} C_VEL
LIN {X 0,Y 481.327,Z 407.637,A -85,B 0,C 180,E1 -6791.075,E2 -6791.075} C_VEL
LIN {X 0,Y 481.432,Z 402.936,A -85,B 0,C 180,E1 -6794.332,E2 -6794.332} C_VEL
LIN {X 0,Y 481.539,Z 399.377,A -85,B 0,C 180,E1 -6796.864,E2 -6796.864} C_VEL
LIN {X 0,Y 481.59,Z 395.946,A -85,B 0,C 180,E1 -6799.362,E2 -6799.362} C_VEL
LIN {X 0,Y 481.606,Z 395.498,A -85,B 0,C 180,E1 -6800.053,E2 -6800.053} C_VEL
LIN {X 0,Y 481.627,Z 395.497,A -85,B 0,C 180,E1 -6802.203,E2 -6802.203} C_VEL
LIN {X 0,Y 481.688,Z 395.49,A -85,B 0,C 180,E1 -6805.318,E2 -6805.318} C_VEL
LIN {X 0,Y 481.643,Z 395.493,A -85,B 0,C 180,E1 -6808.312,E2 -6808.312} C_VEL
LIN {X 0,Y 481.701,Z 395.486,A -85,B 0,C 180,E1 -6811.219,E2 -6811.219} C_VEL
LIN {X 0,Y 481.7,Z 395.485,A -85,B 0,C 180,E1 -6814.043,E2 -6814.043} C_VEL
LIN {X 0,Y 481.668,Z 395.487,A -85,B 0,C 180,E1 -6816.812,E2 -6816.812} C_VEL
LIN {X 0,Y 481.689,Z 395.483,A -85,B 0,C 180,E1 -6819.503,E2 -6819.503} C_VEL
LIN {X 0,Y 481.701,Z 395.482,A -85,B 0,C 180,E1 -6822.158,E2 -6822.158} C_VEL
LIN {X 0,Y 481.736,Z 395.48,A -85,B 0,C 180,E1 -6824.776,E2 -6824.776} C_VEL
LIN {X 0,Y 481.746,Z 395.476,A -85,B 0,C 180,E1 -6828.215,E2 -6828.215} C_VEL
LIN {X 0,Y 481.757,Z 395.475,A -85,B 0,C 180,E1 -6831.612,E2 -6831.612} C_VEL
LIN {X 0,Y 481.81,Z 395.468,A -85,B 0,C 180,E1 -6834.14,E2 -6834.14} C_VEL
LIN {X 0,Y 481.923,Z 395.454,A -85,B 0,C 180,E1 -6837.493,E2 -6837.493} C_VEL
LIN {X 0,Y 481.92,Z 395.457,A -85,B 0,C 180,E1 -6840.836,E2 -6840.836} C_VEL
LIN {X 0,Y 481.922,Z 395.458,A -85,B 0,C 180,E1 -6842.508,E2 -6842.508} C_VEL
LIN {X 0,Y 481.81,Z 395.469,A -85,B 0,C 180,E1 -6845.861,E2 -6845.861} C_VEL
LIN {X 0,Y 481.757,Z 395.475,A -85,B 0,C 180,E1 -6848.389,E2 -6848.389} C_VEL
LIN {X 0,Y 481.789,Z 395.473,A -85,B 0,C 180,E1 -6851.784,E2 -6851.784} C_VEL
LIN {X 0,Y 481.738,Z 395.477,A -85,B 0,C 180,E1 -6855.225,E2 -6855.225} C_VEL
LIN {X 0,Y 481.707,Z 395.484,A -85,B 0,C 180,E1 -6858.722,E2 -6858.722} C_VEL
LIN {X 0,Y 481.641,Z 395.491,A -85,B 0,C 180,E1 -6861.395,E2 -6861.395} C_VEL
LIN {X 0,Y 481.672,Z 395.486,A -85,B 0,C 180,E1 -6864.114,E2 -6864.114} C_VEL
LIN {X 0,Y 481.747,Z 395.477,A -85,B 0,C 180,E1 -6867.141,E2 -6867.141} C_VEL
LIN {X 0,Y 481.684,Z 395.486,A -85,B 0,C 180,E1 -6869.741,E2 -6869.741} C_VEL
LIN {X 0,Y 481.669,Z 395.488,A -85,B 0,C 180,E1 -6872.675,E2 -6872.675} C_VEL
LIN {X 0,Y 481.639,Z 395.49,A -85,B 0,C 180,E1 -6875.71,E2 -6875.71} C_VEL
LIN {X 0,Y 481.668,Z 395.485,A -85,B 0,C 180,E1 -6878.86,E2 -6878.86} C_VEL
LIN {X 0,Y 481.651,Z 395.489,A -85,B 0,C 180,E1 -6881.914,E2 -6881.914} C_VEL
LIN {X 0,Y 481.657,Z 395.491,A -85,B 0,C 180,E1 -6884.458,E2 -6884.458} C_VEL
LIN {X 0,Y 481.652,Z 395.491,A -85,B 0,C 180,E1 -6887.841,E2 -6887.841} C_VEL
LIN {X 0,Y 481.674,Z 395.581,A -85,B 0,C 180,E1 -6890.897,E2 -6890.897} C_VEL
LIN {X 0,Y 482.47,Z 400.166,A -85,B 0,C 180,E1 -6893.329,E2 -6893.329} C_VEL
LIN {X 0,Y 482.614,Z 404.366,A -85,B 0,C 180,E1 -6895.394,E2 -6895.394} C_VEL
LIN {X 0,Y 482.305,Z 410.711,A -85,B 0,C 180,E1 -6898.361,E2 -6898.361} C_VEL
LIN {X 0,Y 482.026,Z 417.168,A -85,B 0,C 180,E1 -6901.24,E2 -6901.24} C_VEL
LIN {X 0,Y 481.713,Z 425.38,A -85,B 0,C 180,E1 -6904.764,E2 -6904.764} C_VEL
LIN {X 0,Y 481.489,Z 433.561,A -85,B 0,C 180,E1 -6908.148,E2 -6908.148} C_VEL
LIN {X 0,Y 481.271,Z 441.312,A -85,B 0,C 180,E1 -6911.261,E2 -6911.261} C_VEL
LIN {X 0,Y 481.122,Z 450.193,A -85,B 0,C 180,E1 -6914.756,E2 -6914.756} C_VEL
LIN {X 0,Y 481.096,Z 450.956,A -85,B 0,C 180,E1 -6915.053,E2 -6915.053} C_VEL
LIN {X 0,Y 483.254,Z 464.761,A -85,B 0,C 180,E1 -6915.485,E2 -6915.485} C_VEL
LIN {X 0,Y 483.87,Z 468.955,A -85,B 0,C 180,E1 -6915.651,E2 -6915.651} C_VEL
LIN {X 0,Y 483.468,Z 481.964,A -85,B 0,C 180,E1 -6916.229,E2 -6916.229} C_VEL
LIN {X 0,Y 483.036,Z 493.158,A -85,B 0,C 180,E1 -6916.892,E2 -6916.892} C_VEL
LIN {X 0,Y 482.642,Z 503.996,A -85,B 0,C 180,E1 -6917.704,E2 -6917.704} C_VEL
LIN {X 0,Y 482.262,Z 514.209,A -85,B 0,C 180,E1 -6918.654,E2 -6918.654} C_VEL
LIN {X 0,Y 481.771,Z 523.394,A -85,B 0,C 180,E1 -6919.706,E2 -6919.706} C_VEL
LIN {X 0,Y 481.429,Z 532.348,A -85,B 0,C 180,E1 -6920.971,E2 -6920.971} C_VEL
LIN {X 0,Y 481.189,Z 539.557,A -85,B 0,C 180,E1 -6922.236,E2 -6922.236} C_VEL
LIN {X 0,Y 480.977,Z 545.402,A -85,B 0,C 180,E1 -6923.522,E2 -6923.522} C_VEL
LIN {X 0,Y 480.9,Z 550.467,A -85,B 0,C 180,E1 -6924.969,E2 -6924.969} C_VEL
LIN {X 0,Y 480.834,Z 552.767,A -85,B 0,C 180,E1 -6925.809,E2 -6925.809} C_VEL
LIN {X 0,Y 480.89,Z 554.634,A -85,B 0,C 180,E1 -6926.649,E2 -6926.649} C_VEL
LIN {X 0,Y 480.793,Z 557.03,A -85,B 0,C 180,E1 -6928.325,E2 -6928.325} C_VEL
LIN {X 0,Y 480.76,Z 557.639,A -85,B 0,C 180,E1 -6929.162,E2 -6929.162} C_VEL
LIN {X 0,Y 480.743,Z 557.857,A -85,B 0,C 180,E1 -6930,E2 -6930} C_VEL
LIN {X 0,Y 480.792,Z 557.039,A -85,B 0,C 180,E1 -6931.675,E2 -6931.675} C_VEL
LIN {X 0,Y 480.823,Z 556.045,A -85,B 0,C 180,E1 -6932.513,E2 -6932.513} C_VEL
LIN {X 0,Y 480.889,Z 554.652,A -85,B 0,C 180,E1 -6933.351,E2 -6933.351} C_VEL
LIN {X 0,Y 480.844,Z 551.715,A -85,B 0,C 180,E1 -6934.611,E2 -6934.611} C_VEL
LIN {X 0,Y 480.956,Z 547.743,A -85,B 0,C 180,E1 -6935.871,E2 -6935.871} C_VEL
LIN {X 0,Y 481.112,Z 541.631,A -85,B 0,C 180,E1 -6937.343,E2 -6937.343} C_VEL
LIN {X 0,Y 481.34,Z 534.952,A -85,B 0,C 180,E1 -6938.607,E2 -6938.607} C_VEL
LIN {X 0,Y 481.665,Z 526.666,A -85,B 0,C 180,E1 -6939.871,E2 -6939.871} C_VEL
LIN {X 0,Y 482.045,Z 518.174,A -85,B 0,C 180,E1 -6940.925,E2 -6940.925} C_VEL
LIN {X 0,Y 482.496,Z 507.68,A -85,B 0,C 180,E1 -6941.979,E2 -6941.979} C_VEL
LIN {X 0,Y 482.865,Z 496.589,A -85,B 0,C 180,E1 -6942.877,E2 -6942.877} C_VEL
LIN {X 0,Y 483.35,Z 485.924,A -85,B 0,C 180,E1 -6943.559,E2 -6943.559} C_VEL
LIN {X 0,Y 483.725,Z 474.244,A -85,B 0,C 180,E1 -6944.138,E2 -6944.138} C_VEL
LIN {X 0,Y 483.658,Z 467.418,A -85,B 0,C 180,E1 -6944.409,E2 -6944.409} C_VEL
LIN {X 0,Y 481.518,Z 453.941,A -85,B 0,C 180,E1 -6944.862,E2 -6944.862} C_VEL
LIN {X 0,Y 481.096,Z 451.04,A -85,B 0,C 180,E1 -6944.947,E2 -6944.947} C_VEL
LIN {X 0,Y 481.213,Z 443.583,A -85,B 0,C 180,E1 -6947.86,E2 -6947.86} C_VEL
LIN {X 0,Y 481.454,Z 435.926,A -85,B 0,C 180,E1 -6950.894,E2 -6950.894} C_VEL
LIN {X 0,Y 481.589,Z 427.968,A -85,B 0,C 180,E1 -6954.117,E2 -6954.117} C_VEL
LIN {X 0,Y 481.817,Z 420.617,A -85,B 0,C 180,E1 -6957.155,E2 -6957.155} C_VEL
LIN {X 0,Y 482.136,Z 413.472,A -85,B 0,C 180,E1 -6960.191,E2 -6960.191} C_VEL
LIN {X 0,Y 482.31,Z 406.787,A -85,B 0,C 180,E1 -6963.122,E2 -6963.122} C_VEL
LIN {X 0,Y 482.505,Z 401.21,A -85,B 0,C 180,E1 -6965.634,E2 -6965.634} C_VEL
LIN {X 0,Y 481.705,Z 395.521,A -85,B 0,C 180,E1 -6968.379,E2 -6968.379} C_VEL
LIN {X 0,Y 481.66,Z 395.491,A -85,B 0,C 180,E1 -6971.04,E2 -6971.04} C_VEL
LIN {X 0,Y 481.679,Z 395.485,A -85,B 0,C 180,E1 -6973.294,E2 -6973.294} C_VEL
LIN {X 0,Y 481.662,Z 395.489,A -85,B 0,C 180,E1 -6976.702,E2 -6976.702} C_VEL
LIN {X 0,Y 481.672,Z 395.485,A -85,B 0,C 180,E1 -6980.059,E2 -6980.059} C_VEL
LIN {X 0,Y 481.624,Z 395.49,A -85,B 0,C 180,E1 -6983.253,E2 -6983.253} C_VEL
LIN {X 0,Y 481.703,Z 395.483,A -85,B 0,C 180,E1 -6986.329,E2 -6986.329} C_VEL
LIN {X 0,Y 481.652,Z 395.486,A -85,B 0,C 180,E1 -6989.415,E2 -6989.415} C_VEL
LIN {X 0,Y 481.694,Z 395.484,A -85,B 0,C 180,E1 -6992.167,E2 -6992.167} C_VEL
LIN {X 0,Y 481.71,Z 395.479,A -85,B 0,C 180,E1 -6994.969,E2 -6994.969} C_VEL
LIN {X 0,Y 481.645,Z 395.49,A -85,B 0,C 180,E1 -6997.704,E2 -6997.704} C_VEL
LIN {X 0,Y 481.697,Z 395.483,A -85,B 0,C 180,E1 -7000.393,E2 -7000.393} C_VEL
LIN {X 0,Y 481.684,Z 395.483,A -85,B 0,C 180,E1 -7003.033,E2 -7003.033} C_VEL
LIN {X 0,Y 481.681,Z 395.486,A -85,B 0,C 180,E1 -7005.638,E2 -7005.638} C_VEL
LIN {X 0,Y 481.742,Z 395.477,A -85,B 0,C 180,E1 -7008.215,E2 -7008.215} C_VEL
LIN {X 0,Y 481.755,Z 395.477,A -85,B 0,C 180,E1 -7011.611,E2 -7011.611} C_VEL
LIN {X 0,Y 481.813,Z 395.467,A -85,B 0,C 180,E1 -7014.139,E2 -7014.139} C_VEL
LIN {X 0,Y 481.92,Z 395.456,A -85,B 0,C 180,E1 -7017.492,E2 -7017.492} C_VEL
LIN {X 0,Y 481.931,Z 395.452,A -85,B 0,C 180,E1 -7020,E2 -7020} C_VEL
LIN {X 0,Y 481.921,Z 395.454,A -85,B 0,C 180,E1 -7022.507,E2 -7022.507} C_VEL
LIN {X 0,Y 481.813,Z 395.467,A -85,B 0,C 180,E1 -7025.86,E2 -7025.86} C_VEL
LIN {X 0,Y 481.755,Z 395.475,A -85,B 0,C 180,E1 -7028.388,E2 -7028.388} C_VEL
LIN {X 0,Y 481.743,Z 395.475,A -85,B 0,C 180,E1 -7031.785,E2 -7031.785} C_VEL
LIN {X 0,Y 481.735,Z 395.478,A -85,B 0,C 180,E1 -7035.224,E2 -7035.224} C_VEL
LIN {X 0,Y 481.703,Z 395.483,A -85,B 0,C 180,E1 -7038.722,E2 -7038.722} C_VEL
LIN {X 0,Y 481.646,Z 395.487,A -85,B 0,C 180,E1 -7041.395,E2 -7041.395} C_VEL
LIN {X 0,Y 481.674,Z 395.487,A -85,B 0,C 180,E1 -7044.113,E2 -7044.113} C_VEL
LIN {X 0,Y 481.744,Z 395.475,A -85,B 0,C 180,E1 -7047.141,E2 -7047.141} C_VEL
LIN {X 0,Y 481.68,Z 395.484,A -85,B 0,C 180,E1 -7049.741,E2 -7049.741} C_VEL
LIN {X 0,Y 481.666,Z 395.485,A -85,B 0,C 180,E1 -7052.675,E2 -7052.675} C_VEL
LIN {X 0,Y 481.636,Z 395.491,A -85,B 0,C 180,E1 -7055.709,E2 -7055.709} C_VEL
LIN {X 0,Y 481.713,Z 395.479,A -85,B 0,C 180,E1 -7059.355,E2 -7059.355} C_VEL
LIN {X 0,Y 481.669,Z 395.485,A -85,B 0,C 180,E1 -7062.158,E2 -7062.158} C_VEL
LIN {X 0,Y 481.654,Z 395.485,A -85,B 0,C 180,E1 -7064.458,E2 -7064.458} C_VEL
LIN {X 0,Y 481.683,Z 395.481,A -85,B 0,C 180,E1 -7066.846,E2 -7066.846} C_VEL
LIN {X 0,Y 481.685,Z 395.482,A -85,B 0,C 180,E1 -7070.062,E2 -7070.062} C_VEL
LIN {X 0,Y 481.626,Z 395.493,A -85,B 0,C 180,E1 -7073.254,E2 -7073.254} C_VEL
LIN {X 0,Y 481.706,Z 395.477,A -85,B 0,C 180,E1 -7076.331,E2 -7076.331} C_VEL
LIN {X 0,Y 481.649,Z 395.49,A -85,B 0,C 180,E1 -7079.418,E2 -7079.418} C_VEL
LIN {X 0,Y 481.7,Z 395.479,A -85,B 0,C 180,E1 -7082.169,E2 -7082.169} C_VEL
LIN {X 0,Y 481.717,Z 395.483,A -85,B 0,C 180,E1 -7084.971,E2 -7084.971} C_VEL
LIN {X 0,Y 481.597,Z 395.492,A -85,B 0,C 180,E1 -7087.99,E2 -7087.99} C_VEL
LIN {X 0,Y 480.887,Z 395.763,A -85,B 0,C 180,E1 -7088.686,E2 -7088.686} C_VEL
LIN {X 0,Y 478.003,Z 397.065,A -85,B 0,C 180,E1 -7089.808,E2 -7089.808} C_VEL
LIN {X 0,Y 475.582,Z 398.516,A -85,B 0,C 180,E1 -7090.707,E2 -7090.707} C_VEL
LIN {X 0,Y 474.543,Z 399.639,A -85,B 0,C 180,E1 -7091.402,E2 -7091.402} C_VEL
LIN {X 0,Y 474.457,Z 399.99,A -85,B 0,C 180,E1 -7091.637,E2 -7091.637} C_VEL
LIN {X 0,Y 474.374,Z 404.221,A -85,B 0,C 180,E1 -7094.534,E2 -7094.534} C_VEL
LIN {X 0,Y 474.321,Z 409.416,A -85,B 0,C 180,E1 -7098.028,E2 -7098.028} C_VEL
LIN {X 0,Y 474.162,Z 414.66,A -85,B 0,C 180,E1 -7101.477,E2 -7101.477} C_VEL
LIN {X 0,Y 474.105,Z 418.608,A -85,B 0,C 180,E1 -7104.044,E2 -7104.044} C_VEL
LIN {X 0,Y 474.098,Z 422.598,A -85,B 0,C 180,E1 -7106.601,E2 -7106.601} C_VEL
LIN {X 0,Y 473.879,Z 426.248,A -85,B 0,C 180,E1 -7108.911,E2 -7108.911} C_VEL
LIN {X 0,Y 476.828,Z 440.997,A -85,B 0,C 180,E1 -7109.446,E2 -7109.446} C_VEL
LIN {X 0,Y 476.99,Z 445.524,A -85,B 0,C 180,E1 -7109.631,E2 -7109.631} C_VEL
LIN {X 0,Y 476.653,Z 457.524,A -85,B 0,C 180,E1 -7110.211,E2 -7110.211} C_VEL
LIN {X 0,Y 476.15,Z 469.166,A -85,B 0,C 180,E1 -7110.952,E2 -7110.952} C_VEL
LIN {X 0,Y 475.655,Z 480.786,A -85,B 0,C 180,E1 -7111.905,E2 -7111.905} C_VEL
LIN {X 0,Y 475.155,Z 491.144,A -85,B 0,C 180,E1 -7112.968,E2 -7112.968} C_VEL
LIN {X 0,Y 474.76,Z 499.541,A -85,B 0,C 180,E1 -7114.032,E2 -7114.032} C_VEL
LIN {X 0,Y 474.402,Z 507.747,A -85,B 0,C 180,E1 -7115.313,E2 -7115.313} C_VEL
LIN {X 0,Y 474.186,Z 515.198,A -85,B 0,C 180,E1 -7116.774,E2 -7116.774} C_VEL
LIN {X 0,Y 473.965,Z 520.447,A -85,B 0,C 180,E1 -7118.098,E2 -7118.098} C_VEL
LIN {X 0,Y 473.805,Z 524.407,A -85,B 0,C 180,E1 -7119.391,E2 -7119.391} C_VEL
LIN {X 0,Y 473.774,Z 526.441,A -85,B 0,C 180,E1 -7120.254,E2 -7120.254} C_VEL
LIN {X 0,Y 473.731,Z 528.929,A -85,B 0,C 180,E1 -7121.724,E2 -7121.724} C_VEL
LIN {X 0,Y 473.655,Z 530.025,A -85,B 0,C 180,E1 -7122.86,E2 -7122.86} C_VEL
LIN {X 0,Y 473.612,Z 530.378,A -85,B 0,C 180,E1 -7123.735,E2 -7123.735} C_VEL
LIN {X 0,Y 473.661,Z 529.978,A -85,B 0,C 180,E1 -7125.325,E2 -7125.325} C_VEL
LIN {X 0,Y 473.622,Z 528.93,A -85,B 0,C 180,E1 -7126.376,E2 -7126.376} C_VEL
LIN {X 0,Y 473.681,Z 527.584,A -85,B 0,C 180,E1 -7127.262,E2 -7127.262} C_VEL
LIN {X 0,Y 473.789,Z 525.39,A -85,B 0,C 180,E1 -7128.314,E2 -7128.314} C_VEL
LIN {X 0,Y 473.938,Z 520.658,A -85,B 0,C 180,E1 -7129.942,E2 -7129.942} C_VEL
LIN {X 0,Y 474.152,Z 515.534,A -85,B 0,C 180,E1 -7131.252,E2 -7131.252} C_VEL
LIN {X 0,Y 474.441,Z 508.533,A -85,B 0,C 180,E1 -7132.652,E2 -7132.652} C_VEL
LIN {X 0,Y 474.783,Z 499.9,A -85,B 0,C 180,E1 -7134.021,E2 -7134.021} C_VEL
LIN {X 0,Y 475.228,Z 490.928,A -85,B 0,C 180,E1 -7135.161,E2 -7135.161} C_VEL
LIN {X 0,Y 475.655,Z 480.734,A -85,B 0,C 180,E1 -7136.207,E2 -7136.207} C_VEL
LIN {X 0,Y 476.209,Z 469.789,A -85,B 0,C 180,E1 -7137.107,E2 -7137.107} C_VEL
LIN {X 0,Y 476.655,Z 458.594,A -85,B 0,C 180,E1 -7137.837,E2 -7137.837} C_VEL
LIN {X 0,Y 477.019,Z 446.63,A -85,B 0,C 180,E1 -7138.431,E2 -7138.431} C_VEL
LIN {X 0,Y 476.951,Z 441.535,A -85,B 0,C 180,E1 -7138.64,E2 -7138.64} C_VEL
LIN {X 0,Y 474.234,Z 428.214,A -85,B 0,C 180,E1 -7139.138,E2 -7139.138} C_VEL
LIN {X 0,Y 473.865,Z 426.331,A -85,B 0,C 180,E1 -7139.224,E2 -7139.224} C_VEL
LIN {X 0,Y 473.964,Z 421.546,A -85,B 0,C 180,E1 -7142.306,E2 -7142.306} C_VEL
LIN {X 0,Y 474.053,Z 416.868,A -85,B 0,C 180,E1 -7145.374,E2 -7145.374} C_VEL
LIN {X 0,Y 474.178,Z 412.208,A -85,B 0,C 180,E1 -7148.498,E2 -7148.498} C_VEL
LIN {X 0,Y 474.297,Z 407.38,A -85,B 0,C 180,E1 -7151.82,E2 -7151.82} C_VEL
LIN {X 0,Y 474.393,Z 403.337,A -85,B 0,C 180,E1 -7154.675,E2 -7154.675} C_VEL
LIN {X 0,Y 474.55,Z 399.053,A -85,B 0,C 180,E1 -7157.772,E2 -7157.772} C_VEL
LIN {X 0,Y 474.557,Z 396.967,A -85,B 0,C 180,E1 -7159.336,E2 -7159.336} C_VEL
LIN {X 0,Y 474.596,Z 396.371,A -85,B 0,C 180,E1 -7160.449,E2 -7160.449} C_VEL
LIN {X 0,Y 474.589,Z 396.375,A -85,B 0,C 180,E1 -7163.677,E2 -7163.677} C_VEL
LIN {X 0,Y 474.638,Z 396.367,A -85,B 0,C 180,E1 -7166.78,E2 -7166.78} C_VEL
LIN {X 0,Y 474.609,Z 396.369,A -85,B 0,C 180,E1 -7169.77,E2 -7169.77} C_VEL
LIN {X 0,Y 474.709,Z 396.356,A -85,B 0,C 180,E1 -7172.681,E2 -7172.681} C_VEL
LIN {X 0,Y 474.653,Z 396.363,A -85,B 0,C 180,E1 -7175.507,E2 -7175.507} C_VEL
LIN {X 0,Y 474.664,Z 396.359,A -85,B 0,C 180,E1 -7179.185,E2 -7179.185} C_VEL
LIN {X 0,Y 474.651,Z 396.362,A -85,B 0,C 180,E1 -7181.884,E2 -7181.884} C_VEL
LIN {X 0,Y 474.693,Z 396.358,A -85,B 0,C 180,E1 -7184.544,E2 -7184.544} C_VEL
LIN {X 0,Y 474.699,Z 396.354,A -85,B 0,C 180,E1 -7188.038,E2 -7188.038} C_VEL
LIN {X 0,Y 474.722,Z 396.351,A -85,B 0,C 180,E1 -7191.487,E2 -7191.487} C_VEL
LIN {X 0,Y 474.773,Z 396.345,A -85,B 0,C 180,E1 -7194.052,E2 -7194.052} C_VEL
LIN {X 0,Y 474.889,Z 396.33,A -85,B 0,C 180,E1 -7197.456,E2 -7197.456} C_VEL
LIN {X 0,Y 474.871,Z 396.335,A -85,B 0,C 180,E1 -7200.848,E2 -7200.848} C_VEL
LIN {X 0,Y 474.889,Z 396.334,A -85,B 0,C 180,E1 -7202.545,E2 -7202.545} C_VEL
LIN {X 0,Y 474.773,Z 396.345,A -85,B 0,C 180,E1 -7205.948,E2 -7205.948} C_VEL
LIN {X 0,Y 474.723,Z 396.353,A -85,B 0,C 180,E1 -7208.514,E2 -7208.514} C_VEL
LIN {X 0,Y 474.732,Z 396.35,A -85,B 0,C 180,E1 -7211.962,E2 -7211.962} C_VEL
LIN {X 0,Y 474.696,Z 396.357,A -85,B 0,C 180,E1 -7215.777,E2 -7215.777} C_VEL
LIN {X 0,Y 474.66,Z 396.363,A -85,B 0,C 180,E1 -7219.011,E2 -7219.011} C_VEL
LIN {X 0,Y 474.585,Z 396.372,A -85,B 0,C 180,E1 -7221.729,E2 -7221.729} C_VEL
LIN {X 0,Y 474.654,Z 396.361,A -85,B 0,C 180,E1 -7224.493,E2 -7224.493} C_VEL
LIN {X 0,Y 474.694,Z 396.355,A -85,B 0,C 180,E1 -7227.339,E2 -7227.339} C_VEL
LIN {X 0,Y 474.606,Z 396.369,A -85,B 0,C 180,E1 -7230.812,E2 -7230.812} C_VEL
LIN {X 0,Y 474.635,Z 396.365,A -85,B 0,C 180,E1 -7233.985,E2 -7233.985} C_VEL
LIN {X 0,Y 474.572,Z 396.372,A -85,B 0,C 180,E1 -7236.901,E2 -7236.901} C_VEL
LIN {X 0,Y 474.625,Z 396.364,A -85,B 0,C 180,E1 -7239.648,E2 -7239.648} C_VEL
LIN {X 0,Y 474.612,Z 396.368,A -85,B 0,C 180,E1 -7242.935,E2 -7242.935} C_VEL
LIN {X 0,Y 474.613,Z 396.369,A -85,B 0,C 180,E1 -7245.896,E2 -7245.896} C_VEL
LIN {X 0,Y 474.631,Z 396.366,A -85,B 0,C 180,E1 -7249.041,E2 -7249.041} C_VEL
LIN {X 0,Y 474.647,Z 396.39,A -85,B 0,C 180,E1 -7250.593,E2 -7250.593} C_VEL
LIN {X 0,Y 475.602,Z 402.304,A -85,B 0,C 180,E1 -7253.767,E2 -7253.767} C_VEL
LIN {X 0,Y 475.572,Z 406.51,A -85,B 0,C 180,E1 -7255.85,E2 -7255.85} C_VEL
LIN {X 0,Y 475.221,Z 413.349,A -85,B 0,C 180,E1 -7259.066,E2 -7259.066} C_VEL
LIN {X 0,Y 474.936,Z 419.281,A -85,B 0,C 180,E1 -7261.737,E2 -7261.737} C_VEL
LIN {X 0,Y 474.638,Z 426.875,A -85,B 0,C 180,E1 -7265.039,E2 -7265.039} C_VEL
LIN {X 0,Y 474.427,Z 434.549,A -85,B 0,C 180,E1 -7268.264,E2 -7268.264} C_VEL
LIN {X 0,Y 474.205,Z 442.563,A -85,B 0,C 180,E1 -7271.536,E2 -7271.536} C_VEL
LIN {X 0,Y 474.047,Z 450.778,A -85,B 0,C 180,E1 -7274.825,E2 -7274.825} C_VEL
LIN {X 0,Y 476.171,Z 464.295,A -85,B 0,C 180,E1 -7275.25,E2 -7275.25} C_VEL
LIN {X 0,Y 476.954,Z 470.225,A -85,B 0,C 180,E1 -7275.493,E2 -7275.493} C_VEL
LIN {X 0,Y 476.581,Z 481.835,A -85,B 0,C 180,E1 -7276.026,E2 -7276.026} C_VEL
LIN {X 0,Y 476.076,Z 494.126,A -85,B 0,C 180,E1 -7276.773,E2 -7276.773} C_VEL
LIN {X 0,Y 475.696,Z 503.416,A -85,B 0,C 180,E1 -7277.486,E2 -7277.486} C_VEL
LIN {X 0,Y 475.26,Z 514.029,A -85,B 0,C 180,E1 -7278.485,E2 -7278.485} C_VEL
LIN {X 0,Y 474.761,Z 523.203,A -85,B 0,C 180,E1 -7279.552,E2 -7279.552} C_VEL
LIN {X 0,Y 474.385,Z 532.148,A -85,B 0,C 180,E1 -7280.836,E2 -7280.836} C_VEL
LIN {X 0,Y 474.108,Z 539.35,A -85,B 0,C 180,E1 -7282.119,E2 -7282.119} C_VEL
LIN {X 0,Y 473.879,Z 545.663,A -85,B 0,C 180,E1 -7283.548,E2 -7283.548} C_VEL
LIN {X 0,Y 473.832,Z 550.26,A -85,B 0,C 180,E1 -7284.894,E2 -7284.894} C_VEL
LIN {X 0,Y 473.74,Z 552.56,A -85,B 0,C 180,E1 -7285.746,E2 -7285.746} C_VEL
LIN {X 0,Y 473.797,Z 554.428,A -85,B 0,C 180,E1 -7286.598,E2 -7286.598} C_VEL
LIN {X 0,Y 473.742,Z 555.826,A -85,B 0,C 180,E1 -7287.449,E2 -7287.449} C_VEL
LIN {X 0,Y 473.688,Z 557.436,A -85,B 0,C 180,E1 -7289.15,E2 -7289.15} C_VEL
LIN {X 0,Y 473.669,Z 557.654,A -85,B 0,C 180,E1 -7290,E2 -7290} C_VEL
LIN {X 0,Y 473.688,Z 557.44,A -85,B 0,C 180,E1 -7290.85,E2 -7290.85} C_VEL
LIN {X 0,Y 473.742,Z 555.842,A -85,B 0,C 180,E1 -7292.551,E2 -7292.551} C_VEL
LIN {X 0,Y 473.797,Z 554.448,A -85,B 0,C 180,E1 -7293.401,E2 -7293.401} C_VEL
LIN {X 0,Y 473.767,Z 551.512,A -85,B 0,C 180,E1 -7294.68,E2 -7294.68} C_VEL
LIN {X 0,Y 473.864,Z 547.538,A -85,B 0,C 180,E1 -7295.959,E2 -7295.959} C_VEL
LIN {X 0,Y 474.032,Z 541.426,A -85,B 0,C 180,E1 -7297.454,E2 -7297.454} C_VEL
LIN {X 0,Y 474.301,Z 534.744,A -85,B 0,C 180,E1 -7298.736,E2 -7298.736} C_VEL
LIN {X 0,Y 474.616,Z 526.45,A -85,B 0,C 180,E1 -7300.02,E2 -7300.02} C_VEL
LIN {X 0,Y 475.036,Z 517.948,A -85,B 0,C 180,E1 -7301.088,E2 -7301.088} C_VEL
LIN {X 0,Y 475.502,Z 507.642,A -85,B 0,C 180,E1 -7302.139,E2 -7302.139} C_VEL
LIN {X 0,Y 475.955,Z 496.042,A -85,B 0,C 180,E1 -7303.089,E2 -7303.089} C_VEL
LIN {X 0,Y 476.47,Z 483.702,A -85,B 0,C 180,E1 -7303.868,E2 -7303.868} C_VEL
LIN {X 0,Y 476.922,Z 471.318,A -85,B 0,C 180,E1 -7304.453,E2 -7304.453} C_VEL
LIN {X 0,Y 475.82,Z 462.174,A -85,B 0,C 180,E1 -7304.815,E2 -7304.815} C_VEL
LIN {X 0,Y 474.035,Z 450.835,A -85,B 0,C 180,E1 -7305.175,E2 -7305.175} C_VEL
LIN {X 0,Y 474.16,Z 443.386,A -85,B 0,C 180,E1 -7308.135,E2 -7308.135} C_VEL
LIN {X 0,Y 474.376,Z 436.194,A -85,B 0,C 180,E1 -7311.035,E2 -7311.035} C_VEL
LIN {X 0,Y 474.555,Z 427.771,A -85,B 0,C 180,E1 -7314.498,E2 -7314.498} C_VEL
LIN {X 0,Y 474.799,Z 420.983,A -85,B 0,C 180,E1 -7317.361,E2 -7317.361} C_VEL
LIN {X 0,Y 475.093,Z 414.405,A -85,B 0,C 180,E1 -7320.195,E2 -7320.195} C_VEL
LIN {X 0,Y 475.295,Z 407.712,A -85,B 0,C 180,E1 -7323.168,E2 -7323.168} C_VEL
LIN {X 0,Y 475.49,Z 402.374,A -85,B 0,C 180,E1 -7325.616,E2 -7325.616} C_VEL
LIN {X 0,Y 474.729,Z 396.852,A -85,B 0,C 180,E1 -7328.314,E2 -7328.314} C_VEL
LIN {X 0,Y 474.671,Z 396.362,A -85,B 0,C 180,E1 -7328.722,E2 -7328.722} C_VEL
LIN {X 0,Y 474.639,Z 396.361,A -85,B 0,C 180,E1 -7332.238,E2 -7332.238} C_VEL
LIN {X 0,Y 474.618,Z 396.364,A -85,B 0,C 180,E1 -7335.296,E2 -7335.296} C_VEL
LIN {X 0,Y 474.624,Z 396.362,A -85,B 0,C 180,E1 -7338.215,E2 -7338.215} C_VEL
LIN {X 0,Y 474.64,Z 396.362,A -85,B 0,C 180,E1 -7340.453,E2 -7340.453} C_VEL
LIN {X 0,Y 474.588,Z 396.366,A -85,B 0,C 180,E1 -7343.676,E2 -7343.676} C_VEL
LIN {X 0,Y 474.637,Z 396.363,A -85,B 0,C 180,E1 -7346.779,E2 -7346.779} C_VEL
LIN {X 0,Y 474.607,Z 396.366,A -85,B 0,C 180,E1 -7349.77,E2 -7349.77} C_VEL
LIN {X 0,Y 474.69,Z 396.356,A -85,B 0,C 180,E1 -7352.679,E2 -7352.679} C_VEL
LIN {X 0,Y 474.651,Z 396.36,A -85,B 0,C 180,E1 -7355.507,E2 -7355.507} C_VEL
LIN {X 0,Y 474.662,Z 396.358,A -85,B 0,C 180,E1 -7359.185,E2 -7359.185} C_VEL
LIN {X 0,Y 474.649,Z 396.362,A -85,B 0,C 180,E1 -7361.884,E2 -7361.884} C_VEL
LIN {X 0,Y 474.691,Z 396.354,A -85,B 0,C 180,E1 -7364.544,E2 -7364.544} C_VEL
LIN {X 0,Y 474.695,Z 396.357,A -85,B 0,C 180,E1 -7368.037,E2 -7368.037} C_VEL
LIN {X 0,Y 474.72,Z 396.353,A -85,B 0,C 180,E1 -7371.486,E2 -7371.486} C_VEL
LIN {X 0,Y 474.775,Z 396.345,A -85,B 0,C 180,E1 -7374.052,E2 -7374.052} C_VEL
LIN {X 0,Y 474.887,Z 396.332,A -85,B 0,C 180,E1 -7377.455,E2 -7377.455} C_VEL
LIN {X 0,Y 474.868,Z 396.335,A -85,B 0,C 180,E1 -7380.848,E2 -7380.848} C_VEL
LIN {X 0,Y 474.887,Z 396.331,A -85,B 0,C 180,E1 -7382.545,E2 -7382.545} C_VEL
LIN {X 0,Y 474.775,Z 396.344,A -85,B 0,C 180,E1 -7385.947,E2 -7385.947} C_VEL
LIN {X 0,Y 474.72,Z 396.353,A -85,B 0,C 180,E1 -7388.514,E2 -7388.514} C_VEL
LIN {X 0,Y 474.696,Z 396.353,A -85,B 0,C 180,E1 -7391.962,E2 -7391.962} C_VEL
LIN {X 0,Y 474.691,Z 396.354,A -85,B 0,C 180,E1 -7395.456,E2 -7395.456} C_VEL
LIN {X 0,Y 474.657,Z 396.36,A -85,B 0,C 180,E1 -7399.01,E2 -7399.01} C_VEL
LIN {X 0,Y 474.589,Z 396.366,A -85,B 0,C 180,E1 -7401.729,E2 -7401.729} C_VEL
LIN {X 0,Y 474.654,Z 396.361,A -85,B 0,C 180,E1 -7404.493,E2 -7404.493} C_VEL
LIN {X 0,Y 474.691,Z 396.353,A -85,B 0,C 180,E1 -7407.339,E2 -7407.339} C_VEL
LIN {X 0,Y 474.602,Z 396.365,A -85,B 0,C 180,E1 -7410.812,E2 -7410.812} C_VEL
LIN {X 0,Y 474.631,Z 396.366,A -85,B 0,C 180,E1 -7413.985,E2 -7413.985} C_VEL
LIN {X 0,Y 474.569,Z 396.368,A -85,B 0,C 180,E1 -7416.901,E2 -7416.901} C_VEL
LIN {X 0,Y 474.649,Z 396.362,A -85,B 0,C 180,E1 -7419.652,E2 -7419.652} C_VEL
LIN {X 0,Y 474.646,Z 396.358,A -85,B 0,C 180,E1 -7422.931,E2 -7422.931} C_VEL
LIN {X 0,Y 474.613,Z 396.365,A -85,B 0,C 180,E1 -7425.897,E2 -7425.897} C_VEL
LIN {X 0,Y 474.641,Z 396.359,A -85,B 0,C 180,E1 -7429.039,E2 -7429.039} C_VEL
LIN {X 0,Y 474.612,Z 396.366,A -85,B 0,C 180,E1 -7431.704,E2 -7431.704} C_VEL
LIN {X 0,Y 474.627,Z 396.36,A -85,B 0,C 180,E1 -7434.727,E2 -7434.727} C_VEL
LIN {X 0,Y 474.635,Z 396.36,A -85,B 0,C 180,E1 -7437.789,E2 -7437.789} C_VEL
LIN {X 0,Y 474.622,Z 396.364,A -85,B 0,C 180,E1 -7440.885,E2 -7440.885} C_VEL
LIN {X 0,Y 474.665,Z 396.357,A -85,B 0,C 180,E1 -7443.629,E2 -7443.629} C_VEL
LIN {X 0,Y 474.634,Z 396.362,A -85,B 0,C 180,E1 -7446.642,E2 -7446.642} C_VEL
LIN {X 0,Y 474.48,Z 396.454,A -85,B 0,C 180,E1 -7449.177,E2 -7449.177} C_VEL
LIN {X 0,Y 474.457,Z 399.99,A -85,B 0,C 180,E1 -7451.637,E2 -7451.637} C_VEL
LIN {X 0,Y 473.783,Z 401.078,A -85,B 0,C 180,E1 -7452.333,E2 -7452.333} C_VEL
LIN {X 0,Y 470.905,Z 403.037,A -85,B 0,C 180,E1 -7453.458,E2 -7453.458} C_VEL
LIN {X 0,Y 468.451,Z 404.624,A -85,B 0,C 180,E1 -7454.364,E2 -7454.364} C_VEL
LIN {X 0,Y 467.366,Z 405.763,A -85,B 0,C 180,E1 -7455.067,E2 -7455.067} C_VEL
LIN {X 0,Y 467.262,Z 406.123,A -85,B 0,C 180,E1 -7455.305,E2 -7455.305} C_VEL
LIN {X 0,Y 467.218,Z 411.177,A -85,B 0,C 180,E1 -7458.724,E2 -7458.724} C_VEL
LIN {X 0,Y 467.069,Z 416.443,A -85,B 0,C 180,E1 -7462.217,E2 -7462.217} C_VEL
LIN {X 0,Y 467.012,Z 420.421,A -85,B 0,C 180,E1 -7464.82,E2 -7464.82} C_VEL
LIN {X 0,Y 467.031,Z 423.092,A -85,B 0,C 180,E1 -7466.549,E2 -7466.549} C_VEL
LIN {X 0,Y 466.772,Z 426.422,A -85,B 0,C 180,E1 -7468.679,E2 -7468.679} C_VEL
LIN {X 0,Y 470.009,Z 442.275,A -85,B 0,C 180,E1 -7469.277,E2 -7469.277} C_VEL
LIN {X 0,Y 469.919,Z 453.564,A -85,B 0,C 180,E1 -7469.786,E2 -7469.786} C_VEL
LIN {X 0,Y 469.362,Z 466.151,A -85,B 0,C 180,E1 -7470.536,E2 -7470.536} C_VEL
LIN {X 0,Y 468.889,Z 477.309,A -85,B 0,C 180,E1 -7471.396,E2 -7471.396} C_VEL
LIN {X 0,Y 468.402,Z 487.389,A -85,B 0,C 180,E1 -7472.365,E2 -7472.365} C_VEL
LIN {X 0,Y 467.91,Z 496.487,A -85,B 0,C 180,E1 -7473.444,E2 -7473.444} C_VEL
LIN {X 0,Y 467.479,Z 505.354,A -85,B 0,C 180,E1 -7474.743,E2 -7474.743} C_VEL
LIN {X 0,Y 467.217,Z 512.5,A -85,B 0,C 180,E1 -7476.044,E2 -7476.044} C_VEL
LIN {X 0,Y 467.008,Z 518.219,A -85,B 0,C 180,E1 -7477.349,E2 -7477.349} C_VEL
LIN {X 0,Y 466.814,Z 522.736,A -85,B 0,C 180,E1 -7478.659,E2 -7478.659} C_VEL
LIN {X 0,Y 466.716,Z 525.123,A -85,B 0,C 180,E1 -7479.535,E2 -7479.535} C_VEL
LIN {X 0,Y 466.685,Z 527.076,A -85,B 0,C 180,E1 -7480.411,E2 -7480.411} C_VEL
LIN {X 0,Y 466.647,Z 529.243,A -85,B 0,C 180,E1 -7481.779,E2 -7481.779} C_VEL
LIN {X 0,Y 466.552,Z 530.347,A -85,B 0,C 180,E1 -7483.059,E2 -7483.059} C_VEL
LIN {X 0,Y 466.516,Z 530.622,A -85,B 0,C 180,E1 -7483.948,E2 -7483.948} C_VEL
LIN {X 0,Y 466.582,Z 530.141,A -85,B 0,C 180,E1 -7485.418,E2 -7485.418} C_VEL
LIN {X 0,Y 466.537,Z 528.857,A -85,B 0,C 180,E1 -7486.632,E2 -7486.632} C_VEL
LIN {X 0,Y 466.614,Z 527.417,A -85,B 0,C 180,E1 -7487.532,E2 -7487.532} C_VEL
LIN {X 0,Y 466.762,Z 524.346,A -85,B 0,C 180,E1 -7488.888,E2 -7488.888} C_VEL
LIN {X 0,Y 466.922,Z 520.108,A -85,B 0,C 180,E1 -7490.254,E2 -7490.254} C_VEL
LIN {X 0,Y 467.126,Z 514.553,A -85,B 0,C 180,E1 -7491.629,E2 -7491.629} C_VEL
LIN {X 0,Y 467.46,Z 507.485,A -85,B 0,C 180,E1 -7493.01,E2 -7493.01} C_VEL
LIN {X 0,Y 467.788,Z 500.166,A -85,B 0,C 180,E1 -7494.167,E2 -7494.167} C_VEL
LIN {X 0,Y 468.256,Z 491.226,A -85,B 0,C 180,E1 -7495.325,E2 -7495.325} C_VEL
LIN {X 0,Y 468.686,Z 481.585,A -85,B 0,C 180,E1 -7496.338,E2 -7496.338} C_VEL
LIN {X 0,Y 469.293,Z 470.175,A -85,B 0,C 180,E1 -7497.298,E2 -7497.298} C_VEL
LIN {X 0,Y 469.782,Z 459.085,A -85,B 0,C 180,E1 -7498.037,E2 -7498.037} C_VEL
LIN {X 0,Y 470.161,Z 447.146,A -85,B 0,C 180,E1 -7498.643,E2 -7498.643} C_VEL
LIN {X 0,Y 470.035,Z 442.253,A -85,B 0,C 180,E1 -7498.853,E2 -7498.853} C_VEL
LIN {X 0,Y 467.379,Z 429.272,A -85,B 0,C 180,E1 -7499.358,E2 -7499.358} C_VEL
LIN {X 0,Y 466.778,Z 426.556,A -85,B 0,C 180,E1 -7499.452,E2 -7499.452} C_VEL
LIN {X 0,Y 466.899,Z 421.824,A -85,B 0,C 180,E1 -7502.548,E2 -7502.548} C_VEL
LIN {X 0,Y 466.994,Z 416.736,A -85,B 0,C 180,E1 -7505.939,E2 -7505.939} C_VEL
LIN {X 0,Y 467.14,Z 411.986,A -85,B 0,C 180,E1 -7509.188,E2 -7509.188} C_VEL
LIN {X 0,Y 467.274,Z 407.136,A -85,B 0,C 180,E1 -7512.595,E2 -7512.595} C_VEL
LIN {X 0,Y 467.377,Z 403.747,A -85,B 0,C 180,E1 -7515.03,E2 -7515.03} C_VEL
LIN {X 0,Y 467.506,Z 400.459,A -85,B 0,C 180,E1 -7517.443,E2 -7517.443} C_VEL
LIN {X 0,Y 467.482,Z 397.451,A -85,B 0,C 180,E1 -7519.726,E2 -7519.726} C_VEL
LIN {X 0,Y 467.558,Z 397.248,A -85,B 0,C 180,E1 -7521.955,E2 -7521.955} C_VEL
LIN {X 0,Y 467.564,Z 397.249,A -85,B 0,C 180,E1 -7525.167,E2 -7525.167} C_VEL
LIN {X 0,Y 467.58,Z 397.245,A -85,B 0,C 180,E1 -7528.26,E2 -7528.26} C_VEL
LIN {X 0,Y 467.578,Z 397.245,A -85,B 0,C 180,E1 -7531.251,E2 -7531.251} C_VEL
LIN {X 0,Y 467.606,Z 397.241,A -85,B 0,C 180,E1 -7534.16,E2 -7534.16} C_VEL
LIN {X 0,Y 467.571,Z 397.245,A -85,B 0,C 180,E1 -7536.996,E2 -7536.996} C_VEL
LIN {X 0,Y 467.616,Z 397.238,A -85,B 0,C 180,E1 -7539.777,E2 -7539.777} C_VEL
LIN {X 0,Y 467.603,Z 397.238,A -85,B 0,C 180,E1 -7542.507,E2 -7542.507} C_VEL
LIN {X 0,Y 467.599,Z 397.238,A -85,B 0,C 180,E1 -7545.196,E2 -7545.196} C_VEL
LIN {X 0,Y 467.65,Z 397.233,A -85,B 0,C 180,E1 -7547.855,E2 -7547.855} C_VEL
LIN {X 0,Y 467.676,Z 397.229,A -85,B 0,C 180,E1 -7551.357,E2 -7551.357} C_VEL
LIN {X 0,Y 467.737,Z 397.222,A -85,B 0,C 180,E1 -7553.963,E2 -7553.963} C_VEL
LIN {X 0,Y 467.854,Z 397.206,A -85,B 0,C 180,E1 -7557.417,E2 -7557.417} C_VEL
LIN {X 0,Y 467.875,Z 397.205,A -85,B 0,C 180,E1 -7560,E2 -7560} C_VEL
LIN {X 0,Y 467.854,Z 397.21,A -85,B 0,C 180,E1 -7562.583,E2 -7562.583} C_VEL
LIN {X 0,Y 467.738,Z 397.221,A -85,B 0,C 180,E1 -7566.038,E2 -7566.038} C_VEL
LIN {X 0,Y 467.676,Z 397.232,A -85,B 0,C 180,E1 -7568.643,E2 -7568.643} C_VEL
LIN {X 0,Y 467.685,Z 397.228,A -85,B 0,C 180,E1 -7572.379,E2 -7572.379} C_VEL
LIN {X 0,Y 467.661,Z 397.234,A -85,B 0,C 180,E1 -7575.893,E2 -7575.893} C_VEL
LIN {X 0,Y 467.619,Z 397.239,A -85,B 0,C 180,E1 -7579.308,E2 -7579.308} C_VEL
LIN {X 0,Y 467.531,Z 397.251,A -85,B 0,C 180,E1 -7582.074,E2 -7582.074} C_VEL
LIN {X 0,Y 467.599,Z 397.244,A -85,B 0,C 180,E1 -7584.888,E2 -7584.888} C_VEL
LIN {X 0,Y 467.624,Z 397.239,A -85,B 0,C 180,E1 -7587.769,E2 -7587.769} C_VEL
LIN {X 0,Y 467.569,Z 397.245,A -85,B 0,C 180,E1 -7591.046,E2 -7591.046} C_VEL
LIN {X 0,Y 467.586,Z 397.241,A -85,B 0,C 180,E1 -7594.243,E2 -7594.243} C_VEL
LIN {X 0,Y 467.547,Z 397.244,A -85,B 0,C 180,E1 -7597.187,E2 -7597.187} C_VEL
LIN {X 0,Y 467.575,Z 397.242,A -85,B 0,C 180,E1 -7600.265,E2 -7600.265} C_VEL
LIN {X 0,Y 467.584,Z 397.243,A -85,B 0,C 180,E1 -7602.568,E2 -7602.568} C_VEL
LIN {X 0,Y 467.568,Z 397.243,A -85,B 0,C 180,E1 -7605.054,E2 -7605.054} C_VEL
LIN {X 0,Y 467.587,Z 397.243,A -85,B 0,C 180,E1 -7607.441,E2 -7607.441} C_VEL
LIN {X 0,Y 467.587,Z 397.244,A -85,B 0,C 180,E1 -7610.299,E2 -7610.299} C_VEL
LIN {X 0,Y 468.439,Z 402.352,A -85,B 0,C 180,E1 -7613.122,E2 -7613.122} C_VEL
LIN {X 0,Y 468.636,Z 406.504,A -85,B 0,C 180,E1 -7615.259,E2 -7615.259} C_VEL
LIN {X 0,Y 468.302,Z 412.83,A -85,B 0,C 180,E1 -7618.315,E2 -7618.315} C_VEL
LIN {X 0,Y 467.977,Z 419.25,A -85,B 0,C 180,E1 -7621.278,E2 -7621.278} C_VEL
LIN {X 0,Y 467.66,Z 426.219,A -85,B 0,C 180,E1 -7624.38,E2 -7624.38} C_VEL
LIN {X 0,Y 467.38,Z 433.346,A -85,B 0,C 180,E1 -7627.453,E2 -7627.453} C_VEL
LIN {X 0,Y 467.198,Z 439.938,A -85,B 0,C 180,E1 -7630.217,E2 -7630.217} C_VEL
LIN {X 0,Y 467.029,Z 447.644,A -85,B 0,C 180,E1 -7633.386,E2 -7633.386} C_VEL
LIN {X 0,Y 466.977,Z 450.525,A -85,B 0,C 180,E1 -7634.557,E2 -7634.557} C_VEL
LIN {X 0,Y 469.42,Z 466.095,A -85,B 0,C 180,E1 -7635.096,E2 -7635.096} C_VEL
LIN {X 0,Y 470.064,Z 471.52,A -85,B 0,C 180,E1 -7635.331,E2 -7635.331} C_VEL
LIN {X 0,Y 469.601,Z 483.747,A -85,B 0,C 180,E1 -7635.925,E2 -7635.925} C_VEL
LIN {X 0,Y 469.018,Z 496.08,A -85,B 0,C 180,E1 -7636.723,E2 -7636.723} C_VEL
LIN {X 0,Y 468.583,Z 507.621,A -85,B 0,C 180,E1 -7637.69,E2 -7637.69} C_VEL
